// TIA Portal project "PHASE2_Final_Team2 Final W HMI" (V16)

(* hardware
DEVICE "S71500/ET200MP station_1"  S7-1500 station
   slot 0: "Rail_0"  Rack  6ES7 590-1***0-0AA0
   slot 1: "PLC_1"  CPU 1513-1 PN  6ES7 513-1AL02-0AB0  V2.8
      slot 3: "CPU display_1"  6ES7591-1AA00-0AA0
      slot 32768: "PROFINET interface_1"  X1
         slot 32769: "Port_1"  X1 P1
         slot 32770: "Port_2"  X1 P2
      slot 34817: "Virtual CP interface port_1"  Virtual CP interface port  Virtual CP interface port
   slot 2: "DI 16x24VDC BA_1"  DI 16x24VDC BA  6ES7 521-1BH10-0AA0  V1.1
   slot 3: "DQ 16x24VDC/0.5A BA_1"  DQ 16x24VDC/0.5A BA  6ES7 522-1BH10-0AA0  V1.1
DEVICE "HMI_1"  TP700 Comfort
   slot 0: "HMI_1"  TP700 Comfort  6AV2 124-0GC01-0AX0  16.0.0.0
   slot 1: "HMI_RT_1"  TP700 Comfort  6AV2 124-0GC01-0AX0  16.0.0.0
   slot 5: "HMI_1.IE_CP_1"  PROFINET Interface  16.0.0.0
      slot 1: "PROFINET Interface_1"  PROFINET Interface
         slot 1: "Port_1"  Port
         slot 2: "Port_2"  Port
   slot 7: "HMI_1.MPI/DP_CP_1"  MPI/DP Interface  16.0.0.0
*)

// ===== PLC "PLC_1"  CPU 1513-1 PN =====

VAR_GLOBAL   // PLC tag table "Default tag table"
   "start whole system" AT %I3.1 : Bool;
   "stop whole system" AT %I3.2 : Bool;
   "Lid Exit Stop" AT %M251.0 : Bool;
   "LID exit Stop Sensor" AT %I7.2 : Bool;
   "Base Exit Stop Sensor" AT %I7.1 : Bool;
   "Base Exit Stop" AT %M250.0 : Bool;
END_VAR

VAR_GLOBAL   // PLC tag table "pick&place"
   "Item_at_entry" AT %I0.0 : Bool;
   "Item at Exit" AT %I0.1 : Bool;
   "Moving X" AT %M171.0 : Bool;
   "Moving Z" AT %M170.0 : Bool;
   "Item Detected" AT %I0.2 : Bool;
   "Start Button" AT %I0.3 : Bool;
   "Reset" AT %I0.4 : Bool;
   "Stop" AT %I0.5 : Bool;
   "Emergency stop" AT %I0.6 : Bool;
   "Entry_conveyor" AT %Q5.0 : Bool;
   "Exit conveyor" AT %Q5.1 : Bool;
   "Move X" AT %Q5.2 : Bool;
   "Move Z" AT %Q12.3 : Bool;
   "Grab" AT %Q0.4 : Bool;
   "Start light 1" AT %Q4.5 : Bool;
   "Reset light 1" AT %Q5.6 : Bool;
   "Stop light 1" AT %Q0.7 : Bool;
   "s1" AT %M92.0 : Bool;
   "s2" AT %M93.0 : Bool;
   "s3" AT %M94.0 : Bool;
   "s4" AT %M95.0 : Bool;
   "s5" AT %M96.0 : Bool;
   "s6" AT %M97.0 : Bool;
   "s7" AT %M98.0 : Bool;
   "s8" AT %M99.0 : Bool;
   "Entry Conveyor 1" AT %QD30 : Real;
   "Exit_Conveyor 1" AT %QD34 : Real;
   "Move_X 1" AT %QD38 : Real;
   "Move_Z 1" AT %QD42 : Real;
   "Moving_X 1" AT %ID30 : Real;
   "Moving_Z 1" AT %ID34 : Real;
   "Item_at_entry(1)" AT %I0.7 : Bool;
   "Item at Exit(1)" AT %I1.0 : Bool;
   "Moving X(1)" AT %M172.0 : Bool;
   "Moving Z(1)" AT %M173.0 : Bool;
   "Item Detected(1)" AT %I1.1 : Bool;
   "Start Button(1)" AT %I1.2 : Bool;
   "Reset(1)" AT %I1.3 : Bool;
   "Stop(1)" AT %I1.4 : Bool;
   "Emergency stop(1)" AT %I1.5 : Bool;
   "Entry_conveyor(1)" AT %M120.0 : Bool;
   "Exit conveyor(1)" AT %Q7.1 : Bool;
   "Move X(1)" AT %Q7.2 : Bool;
   "Move Z(1)" AT %Q7.3 : Bool;
   "Grab(1)" AT %Q0.5 : Bool;
   "Start light 1(1)" AT %Q3.5 : Bool;
   "Reset light 1(1)" AT %Q3.6 : Bool;
   "Stop light 1(1)" AT %Q3.7 : Bool;
   "Counter 1(1)" AT %QD60 : DInt;
   "s1(1)" AT %M14.0 : Bool;
   "s2(1)" AT %M101.0 : Bool;
   "s3(1)" AT %M102.0 : Bool;
   "s4(1)" AT %M103.0 : Bool;
   "s5(1)" AT %M104.0 : Bool;
   "s6(1)" AT %M105.0 : Bool;
   "s7(1)" AT %M106.0 : Bool;
   "s8(1)" AT %M107.0 : Bool;
   "Entry Conveyor 1(1)" AT %QD46 : Real;
   "Exit_Conveyor 1(1)" AT %QD50 : Real;
   "Move_X 1(1)" AT %QD54 : Real;
   "Move_Z 1(1)" AT %QD58 : Real;
   "Moving_X 1(1)" AT %ID38 : Real;
   "Moving_Z 1(1)" AT %ID42 : Real;
   "Emitter 1" AT %Q2.2 : Bool;
   "Emitter 0" AT %Q2.3 : Bool;
END_VAR

VAR_GLOBAL   // PLC tag table "machine_center"
   "Start_System" AT %I2.6 : Bool;
   "Stop_System" AT %I2.7 : Bool;
   "Lids_Raw_conveyor" AT %M72.0 : Bool;
   "Bases_raw_conveyor" AT %M73.0 : Bool;
   "S1(2)" AT %M100.0 : Bool;
   "S2(2)" AT %M108.0 : Bool;
   "S3(2)" AT %M109.0 : Bool;
   "S4(2)" AT %M110.0 : Bool;
   "S5(2)" AT %M111.0 : Bool;
   "S6(2)" AT %M112.0 : Bool;
   "S7(2)" AT %M113.0 : Bool;
   "S8(2)" AT %M8.0 : Bool;
   "S9" AT %M9.0 : Bool;
   "S10" AT %M10.0 : Bool;
   "Emergency Stop System" AT %I3.0 : Bool;
   "Start_Light" AT %Q1.1 : Bool;
   "Stop_lights" AT %Q1.2 : Bool;
   "Lids_at_entry" AT %I1.6 : Bool;
   "Bases At entry" AT %I2.2 : Bool;
   "Lids_center_busy" AT %I1.7 : Bool;
   "Lids_at_exit" AT %I2.1 : Bool;
   "Lids_center_error" AT %I2.0 : Bool;
   "Bases_at_exit" AT %I2.5 : Bool;
   "bases_center_busy" AT %I2.3 : Bool;
   "Base_center_error" AT %I2.4 : Bool;
   "S11" AT %M11.0 : Bool;
   "S12" AT %M12.0 : Bool;
   "Exit_Conveyor" AT %Q11.6 : Bool;
   "Produce_Lids" AT %Q0.0 : Bool;
   "Lids_Center_Start" AT %Q0.1 : Bool;
   "Bases_center_start" AT %Q0.6 : Bool;
   "Reset_Lids" AT %Q0.2 : Bool;
   "Stop_Lids" AT %Q0.3 : Bool;
   "Reset_Base" AT %Q10.6 : Bool;
   "Stop_Bases" AT %Q10.7 : Bool;
   "Lids_Exit_convyor1" AT %M70.0 : Bool;
   "LIDS Sorting Conveyor1" AT %M71.0 : Bool;
   "Bases_Exit_conveyor1" AT %M206.0 : Bool;
   "Bases Sorting Conveyor" AT %M205.0 : Bool;
   "Lids_Count" AT %QW10 : Int;
   "Bases_Count" AT %QW20 : Int;
   "Tag_1" AT %M13.0 : Bool;
   "S13" AT %M64.0 : Bool;
   "S14" AT %M65.0 : Bool;
   "Tag_2" AT %M66.0 : Bool;
   "Tag_3" AT %M67.0 : Bool;
   "Lids_Arrived" AT %I11.5 : Bool;
   "Bases Arrived" AT %I11.4 : Bool;
   "LIDS_RAW_CONVEYOR_aNALOG" AT %QD62 : Real;
   "Lid_exit_conveyor1_analog" AT %QD66 : Real;
   "Base_raw_conveyor_analog" AT %QD70 : Real;
   "Base_exit_conveyor1_analog" AT %QD74 : Real;
END_VAR

VAR_GLOBAL   // PLC tag table "Sorting"
   "Bases Sorter turn" AT %Q1.5 : Bool;
   "bases Sorter  Belt" AT %Q1.6 : Bool;
   "LID sorter Turn" AT %Q1.3 : Bool;
   "LID sorter Belt" AT %Q1.4 : Bool;
   "Base Sorting Sensor" AT %ID50 : DWord;
   "Base_Exit_conveyor_blue" AT %M84.0 : Bool;
   "Vision sensor in range" AT %Q46.4 : Bool;
   "Stop Entry conveyor" AT %Q46.5 : Bool;
   "Blue lid" AT %M200.0 : Bool;
   "Green lid" AT %M201.0 : Bool;
   "Tag_1(1)" AT %M50.0 : Bool;
   "Tag_2(1)" AT %M51.0 : Bool;
   "S1(3)" AT %M52.0 : Bool;
   "S2(3)" AT %M53.0 : Bool;
   "S3(3)" AT %M54.0 : Bool;
   "S4(3)" AT %M55.0 : Bool;
   "S5(3)" AT %M56.0 : Bool;
   "S6(3)" AT %M57.0 : Bool;
   "S1(4)" AT %M58.0 : Bool;
   "S2(4)" AT %M59.0 : Bool;
   "S3(4)" AT %M60.0 : Bool;
   "S5(4)" AT %M61.0 : Bool;
   "S4(4)" AT %M62.0 : Bool;
   "S6(4)" AT %M63.0 : Bool;
   "Base Start Sorting" AT %I4.0 : Bool;
   "Base Exit Conveyor Green" AT %M85.0 : Bool;
   "Bases Blue Sorted Conv" AT %QD106 : Real;
   "Bases Green Sorted Conv" AT %QD102 : Real;
   "LID Start Sorting" AT %I3.7 : Bool;
   "LID sorting Sensor" AT %ID46 : DWord;
   "LIDs_Blue_Sorted_conv" AT %M86.0 : Bool;
   "LIDs green sorted conv" AT %M87.0 : Bool;
   "LID blue sorted conv ana" AT %QD98 : Real;
   "LID green Sorted Conv ANalog" AT %QD94 : Real;
   "Emergency Stop Base" AT %I4.1 : Bool;
   "Emergency Stop LID" AT %I4.2 : Bool;
   "Blue Base" AT %M90.0 : Bool;
   "Green Base" AT %M91.0 : Bool;
   "LID Green Sorted" AT %I3.4 : Bool;
   "LID Blue Sorted" AT %I3.3 : Bool;
   "LIDS sorting Conveyor 2" AT %M82.0 : Bool;
   "Base Blue Sorted" AT %I3.5 : Bool;
   "Base Green Sorted" AT %I3.6 : Bool;
   "Curved Bases Sorting Conveyor" AT %M83.0 : Bool;
   "LID sorting conveyor 1" AT %QD78 : Real;
   "LID Sorting Conveyor 2" AT %QD82 : Real;
   "Base Sorting Conveyor" AT %QD86 : Real;
   "Curved Base Sorting Conveyor" AT %QD90 : Real;
   "LID green Sorted Conv ANalog(1)" AT %QD110 : Real;
   "LID green Sorted Conv ANalog(2)" AT %QD114 : Real;
   "LID green Sorted Conv ANalog(3)" AT %QD118 : Real;
   "LID blue sorted conv ana(1)" AT %QD122 : Real;
   "LID blue sorted conv ana(2)" AT %QD126 : Real;
   "Bases Blue Sorted Conv(1)" AT %QD130 : Real;
   "Bases Blue Sorted Conv(2)" AT %QD134 : Real;
   "Bases Green Sorted Conv(1)" AT %QD138 : Real;
   "Bases Green Sorted Conv(2)" AT %QD142 : Real;
   "Bases Green Sorted Conv(3)" AT %QD146 : Real;
   "Bases Green Sorted Conv(4)" AT %QD150 : Real;
   "Bases Green Sorted Conv(5)" AT %QD154 : Real;
   "Bases Green Sorted Conv(6)" AT %QD158 : Real;
END_VAR

VAR_GLOBAL   // PLC tag table "BlueAssembler"
   "S1(7) Blue Assembler" AT %M121.0 : Bool;
   "S2(7) Blue Assembler" AT %M122.0 : Bool;
   "S3(7) Blue Assembler" AT %M123.0 : Bool;
   "S4(7) Blue Assembler" AT %M124.0 : Bool;
   "S5(7) Blue Assembler" AT %M125.0 : Bool;
   "S6(7) Blue Assembler" AT %M126.0 : Bool;
   "S7(5) Blue Assembler" AT %M127.0 : Bool;
   "S8(5) Blue Assembler" AT %M128.0 : Bool;
   "S9(1) Blue Assembler" AT %M129.0 : Bool;
   "Emergency Stop Blue Assembler" AT %I5.3 : Bool;
   "Lid at place Blue Assembler" AT %I4.6 : Bool;
   "base at place Blue Assembler" AT %I5.0 : Bool;
   "Lid_clamped Blue Assembler" AT %I4.7 : Bool;
   "Item Detected Blue Assembler" AT %I4.5 : Bool;
   "Moving_z Blue Assembler" AT %I4.4 : Bool;
   "Tag_1(2) Blue Assembler" AT %M139.0 : Bool;
   "Base Clamped Blue Assembler" AT %I5.1 : Bool;
   "Tag_2(2) Blue Assembler" AT %M140.0 : Bool;
   "Moving_X Blue Assembler" AT %I4.3 : Bool;
   "Tag_3(1) Blue Assembler" AT %M141.0 : Bool;
   "Tag_4 Blue Assembler" AT %M142.0 : Bool;
   "Part_leaving Blue Assembler" AT %I5.2 : Bool;
   "S10(1) Blue Assembler" AT %M143.0 : Bool;
   "Tag_5 Blue Assembler" AT %M144.0 : Bool;
   "Lid _ Conveyor Blue Assembler" AT %M151.0 : Bool;
   "Bases Conveyor Blue Assembler" AT %M152.0 : Bool;
   "Clamp-base Blue Assembler" AT %Q2.5 : Bool;
   "Clamp_lid Blue Assembler" AT %Q2.6 : Bool;
   "grab Blue Assembler" AT %Q2.4 : Bool;
   "Pos_raise_bases Blue Assembler" AT %Q2.7 : Bool;
   "Tag_6Blue Assembler" AT %M147.0 : Bool;
   "S11(1) Blue Assembler" AT %M150.0 : Bool;
   "Tag_7Blue Assembler" AT %M145.0 : Bool;
   "Tag_8Blue Assembler" AT %M146.0 : Bool;
   "Lid_Conveyor_Analog Blue Assembler" AT %QD162 : Real;
   "Base_Conveyor_analog Blue Assembler" AT %QD166 : Real;
   "move_xBlue Assembler" AT %M148.0 : Bool;
   "Move_X_analog Blue Assembler" AT %QD170 : Real;
   "move_z Blue Assembler" AT %M149.0 : Bool;
   "Move_Z_analog Blue Assembler" AT %QD174 : Real;
   "Start base BlueAssembly(1)" AT %I5.4 : Bool;
   "Start LID Blue Assembly(1)" AT %I5.5 : Bool;
END_VAR

VAR_GLOBAL   // PLC tag table "GreenAssembler"
   "S1(8) Green" AT %M130.0 : Bool;
   "S2(8) Green" AT %M131.0 : Bool;
   "S3(8) Green" AT %M132.0 : Bool;
   "S4(8) Green" AT %M133.0 : Bool;
   "S5(8) Green" AT %M134.0 : Bool;
   "S6(8) Green" AT %M135.0 : Bool;
   "S7(6) Green" AT %M136.0 : Bool;
   "S8(6) Green" AT %M137.0 : Bool;
   "S9(2) Green" AT %M138.0 : Bool;
   "Emergency Stop Green assembler" AT %I6.6 : Bool;
   "Lid at place(1) Green" AT %I6.1 : Bool;
   "base at place(1) Green" AT %I6.3 : Bool;
   "Lid_clamped(1) Green" AT %I6.2 : Bool;
   "Item Detected(3) Green" AT %I6.0 : Bool;
   "Moving_z(1) Green" AT %I5.7 : Bool;
   "Tag_1(3) Green" AT %M153.0 : Bool;
   "Base Clamped(1) Green" AT %I6.4 : Bool;
   "Tag_2(3) Green" AT %M154.0 : Bool;
   "Moving_X Green" AT %I5.6 : Bool;
   "Tag_3(2) Green" AT %M155.0 : Bool;
   "Tag_4(1) Green" AT %M156.0 : Bool;
   "Part_leaving(1) Green" AT %I6.5 : Bool;
   "S10(2) Green" AT %M157.0 : Bool;
   "Tag_5(1) Green" AT %M158.0 : Bool;
   "Lid _ Conveyor(1) Green" AT %M165.0 : Bool;
   "Bases Conveyor(1) Green" AT %M166.0 : Bool;
   "Clamp-base(1) Green" AT %Q3.1 : Bool;
   "Clamp_lid(1) Green" AT %Q3.2 : Bool;
   "grab(4) Green" AT %Q3.0 : Bool;
   "Pos_raise_bases(1) Green" AT %Q3.3 : Bool;
   "Tag_6(1) Green" AT %M161.0 : Bool;
   "S11(2) Green" AT %M164.0 : Bool;
   "Tag_7(1) Green" AT %M159.0 : Bool;
   "Tag_8(1) Green" AT %M160.0 : Bool;
   "Lid_Conveyor_Analog(1) Green" AT %QD178 : Real;
   "Base_Conveyor_analog(1) Green" AT %QD182 : Real;
   "move_x(1) Green" AT %M162.0 : Bool;
   "Move_X_analog(1) Green" AT %QD186 : Real;
   "move_z(1) Green" AT %M163.0 : Bool;
   "Move_Z_analog(1) Green" AT %QD190 : Real;
   "Start base Green Assembly" AT %I6.7 : Bool;
   "Start LID Green Assembly" AT %I7.0 : Bool;
END_VAR

DATA_BLOCK "machine_center_DB"   // DB1
{ S7_Optimized_Access := 'TRUE' }
VERSION : 0.1
// stored: InstanceOfName machine_center
"machine_center"
BEGIN
END_DATA_BLOCK

DATA_BLOCK "Sorting2_DB"   // DB2
{ S7_Optimized_Access := 'TRUE' }
VERSION : 0.1
// stored: InstanceOfName Sorting2
"Sorting2"
BEGIN
END_DATA_BLOCK

DATA_BLOCK "Pick&Place1_DB"   // DB3
{ S7_Optimized_Access := 'TRUE' }
VERSION : 0.1
// stored: InstanceOfName Pick&Place1
"Pick&Place1"
BEGIN
END_DATA_BLOCK

DATA_BLOCK "Pick&Place2_DB"   // DB4
{ S7_Optimized_Access := 'TRUE' }
VERSION : 0.1
// stored: InstanceOfName Pick&Place2
"Pick&Place2"
BEGIN
END_DATA_BLOCK

DATA_BLOCK "Sorting1_DB"   // DB5
{ S7_Optimized_Access := 'TRUE' }
VERSION : 0.1
// stored: InstanceOfName Sorting1
"Sorting1"
BEGIN
END_DATA_BLOCK

DATA_BLOCK "Assembler Blue_DB"   // DB6
{ S7_Optimized_Access := 'TRUE' }
VERSION : 0.1
// stored: InstanceOfName Assembler Blue
"Assembler Blue"
BEGIN
END_DATA_BLOCK

DATA_BLOCK "Assembler Green_DB"   // DB7
{ S7_Optimized_Access := 'TRUE' }
VERSION : 0.1
// stored: InstanceOfName Assembler Green
"Assembler Green"
BEGIN
END_DATA_BLOCK

DATA_BLOCK "HMI_Area_Pointer"   // DB8
{ S7_Optimized_Access := 'TRUE' }
VERSION : 0.1
   VAR
      "Job MailBox" : Array[0..3] of Word;
      NumScreen : Int;
      "Start Whole System PB" : Bool;
      "Stop Whole System PB" : Bool;
      HMI_Box_Pick_and_place1 : DWord := 0;
      HMI_Box_Pick_and_place2 : DWord := 0;
      "HMI blue part sorted move HMI" : DWord := 0;
      "HMI Green part sorted move HMI" : DWord := 0;
   END_VAR
BEGIN
   "Job MailBox"[0] := 51;
   "Job MailBox"[2] := 0;
   "Job MailBox"[3] := 0;
END_DATA_BLOCK

// folder: System blocks/Program resources

DATA_BLOCK "IEC_Timer_0_DB"   // DB9
{ S7_Optimized_Access := 'TRUE' }
AUTHOR : Simatic
FAMILY : IEC
NAME : IEC_TMR
VERSION : 1.0
// stored: InstanceOfName IEC_TIMER
"IEC_TIMER"
BEGIN
END_DATA_BLOCK

DATA_BLOCK "IEC_Timer_0_DB_1"   // DB10
{ S7_Optimized_Access := 'TRUE' }
AUTHOR : Simatic
FAMILY : IEC
NAME : IEC_TMR
VERSION : 1.0
// stored: InstanceOfName IEC_TIMER
"IEC_TIMER"
BEGIN
END_DATA_BLOCK

DATA_BLOCK "IEC_Timer_0_DB_2"   // DB11
{ S7_Optimized_Access := 'TRUE' }
AUTHOR : Simatic
FAMILY : IEC
NAME : IEC_TMR
VERSION : 1.0
// stored: InstanceOfName IEC_TIMER
"IEC_TIMER"
BEGIN
END_DATA_BLOCK

DATA_BLOCK "IEC_Timer_0_DB_3"   // DB12
{ S7_Optimized_Access := 'TRUE' }
AUTHOR : Simatic
FAMILY : IEC
NAME : IEC_TMR
VERSION : 1.0
// stored: InstanceOfName IEC_TIMER
"IEC_TIMER"
BEGIN
END_DATA_BLOCK

// folder: (top level)

FUNCTION_BLOCK "Pick&Place1"   // FB1, LAD
{ S7_Optimized_Access := 'TRUE' }
VERSION : 0.1
BEGIN

REGION Network 1
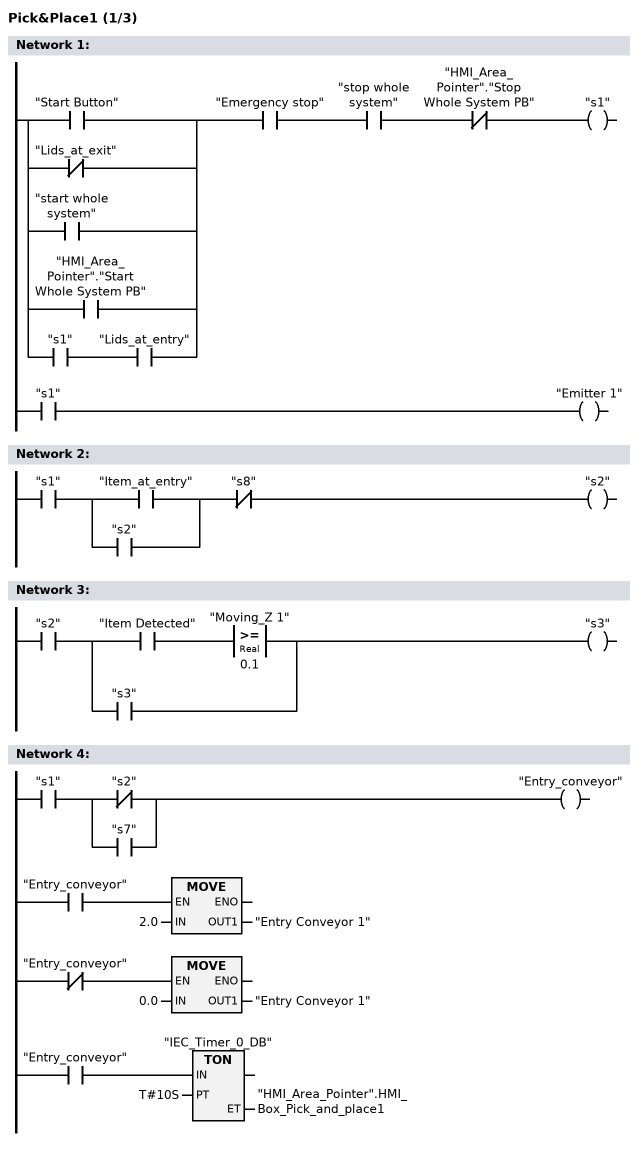
   RUNG wire#powerrail
      Contact( "Start Button" )
      wire#w1
      Contact( "Emergency stop" )
      Contact( "stop whole system" )
      I_Contact( "HMI_Area_Pointer"."Stop Whole System PB" )
      Coil( "s1" )
   END_RUNG
   RUNG wire#powerrail
      I_Contact( "Lids_at_exit" )
   END_RUNG wire#w1
   RUNG wire#powerrail
      Contact( "start whole system" )
   END_RUNG wire#w1
   RUNG wire#powerrail
      Contact( "HMI_Area_Pointer"."Start Whole System PB" )
   END_RUNG wire#w1
   RUNG wire#powerrail
      Contact( "s1" )
      Contact( "Lids_at_entry" )
   END_RUNG wire#w1
   RUNG wire#powerrail
      Contact( "s1" )
      Coil( "Emitter 1" )
   END_RUNG
   // the same network as SCL:
   "s1" := ("Start Button" OR NOT "Lids_at_exit" OR "start whole system" OR "HMI_Area_Pointer"."Start Whole System PB" OR ("s1" AND "Lids_at_entry")) AND "Emergency stop" AND "stop whole system" AND NOT "HMI_Area_Pointer"."Stop Whole System PB";
   "Emitter 1" := "s1";
END_REGION

REGION Network 2
   RUNG wire#powerrail
      Contact( "s1" )
      wire#w1
      Contact( "Item_at_entry" )
      wire#w2
      I_Contact( "s8" )
      Coil( "s2" )
   END_RUNG
   RUNG wire#w1
      Contact( "s2" )
   END_RUNG wire#w2
   // the same network as SCL:
   "s2" := "s1" AND ("Item_at_entry" OR "s2") AND NOT "s8";
END_REGION

REGION Network 3
   RUNG wire#powerrail
      Contact( "s2" )
      wire#w1
      Contact( "Item Detected" )
      { S7_Templates := "SrcType := Real" } GE_Contact(in1 := "Moving_Z 1", in2 := 0.1)
      wire#w2
      Coil( "s3" )
   END_RUNG
   RUNG wire#w1
      Contact( "s3" )
   END_RUNG wire#w2
   // the same network as SCL:
   "s3" := "s2" AND (("Item Detected" AND ("Moving_Z 1" >= 0.1)) OR "s3");
END_REGION

REGION Network 4
   "Entry_conveyor" := "s1" AND (NOT "s2" OR "s7");
   IF "Entry_conveyor" THEN "Entry Conveyor 1" := 2.0; END_IF;
   IF NOT "Entry_conveyor" THEN "Entry Conveyor 1" := 0.0; END_IF;
   "IEC_Timer_0_DB".TON(IN := "Entry_conveyor", PT := T#10S, ET => "HMI_Area_Pointer".HMI_Box_Pick_and_place1);
END_REGION

REGION Network 5
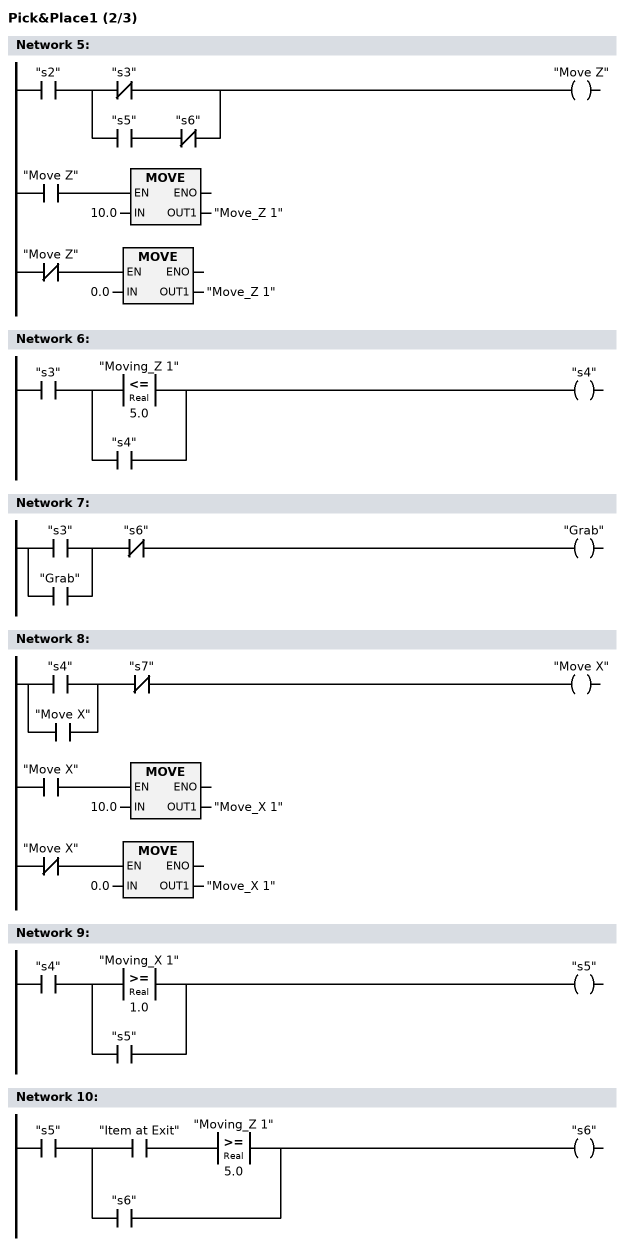
   RUNG wire#powerrail
      Contact( "s2" )
      wire#w1
      I_Contact( "s3" )
      wire#w2
      Coil( "Move Z" )
   END_RUNG
   RUNG wire#w1
      Contact( "s5" )
      I_Contact( "s6" )
   END_RUNG wire#w2
   RUNG wire#powerrail
      Contact( "Move Z" )
      Move(in := 10.0, out1 => "Move_Z 1")
   END_RUNG
   RUNG wire#powerrail
      I_Contact( "Move Z" )
      Move(in := 0.0, out1 => "Move_Z 1")
   END_RUNG
   // the same network as SCL:
   "Move Z" := "s2" AND (NOT "s3" OR ("s5" AND NOT "s6"));
   IF "Move Z" THEN "Move_Z 1" := 10.0; END_IF;
   IF NOT "Move Z" THEN "Move_Z 1" := 0.0; END_IF;
END_REGION

REGION Network 6
   RUNG wire#powerrail
      Contact( "s3" )
      wire#w1
      { S7_Templates := "SrcType := Real" } LE_Contact(in1 := "Moving_Z 1", in2 := 5.0)
      wire#w2
      Coil( "s4" )
   END_RUNG
   RUNG wire#w1
      Contact( "s4" )
   END_RUNG wire#w2
   // the same network as SCL:
   "s4" := "s3" AND (("Moving_Z 1" <= 5.0) OR "s4");
END_REGION

REGION Network 7
   RUNG wire#powerrail
      Contact( "s3" )
      wire#w1
      I_Contact( "s6" )
      Coil( "Grab" )
   END_RUNG
   RUNG wire#powerrail
      Contact( "Grab" )
   END_RUNG wire#w1
   // the same network as SCL:
   "Grab" := ("s3" OR "Grab") AND NOT "s6";
END_REGION

REGION Network 8
   RUNG wire#powerrail
      Contact( "s4" )
      wire#w1
      I_Contact( "s7" )
      Coil( "Move X" )
   END_RUNG
   RUNG wire#powerrail
      Contact( "Move X" )
   END_RUNG wire#w1
   RUNG wire#powerrail
      Contact( "Move X" )
      Move(in := 10.0, out1 => "Move_X 1")
   END_RUNG
   RUNG wire#powerrail
      I_Contact( "Move X" )
      Move(in := 0.0, out1 => "Move_X 1")
   END_RUNG
   // the same network as SCL:
   "Move X" := ("s4" OR "Move X") AND NOT "s7";
   IF "Move X" THEN "Move_X 1" := 10.0; END_IF;
   IF NOT "Move X" THEN "Move_X 1" := 0.0; END_IF;
END_REGION

REGION Network 9
   RUNG wire#powerrail
      Contact( "s4" )
      wire#w1
      { S7_Templates := "SrcType := Real" } GE_Contact(in1 := "Moving_X 1", in2 := 1.0)
      wire#w2
      Coil( "s5" )
   END_RUNG
   RUNG wire#w1
      Contact( "s5" )
   END_RUNG wire#w2
   // the same network as SCL:
   "s5" := "s4" AND (("Moving_X 1" >= 1.0) OR "s5");
END_REGION

REGION Network 10
   RUNG wire#powerrail
      Contact( "s5" )
      wire#w1
      Contact( "Item at Exit" )
      { S7_Templates := "SrcType := Real" } GE_Contact(in1 := "Moving_Z 1", in2 := 5.0)
      wire#w2
      Coil( "s6" )
   END_RUNG
   RUNG wire#w1
      Contact( "s6" )
   END_RUNG wire#w2
   // the same network as SCL:
   "s6" := "s5" AND (("Item at Exit" AND ("Moving_Z 1" >= 5.0)) OR "s6");
END_REGION

REGION Network 11
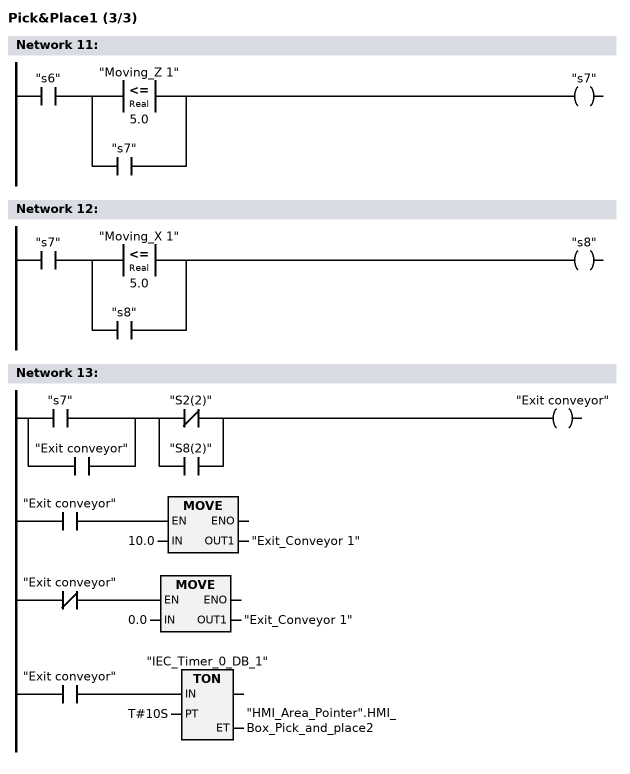
   RUNG wire#powerrail
      Contact( "s6" )
      wire#w1
      { S7_Templates := "SrcType := Real" } LE_Contact(in1 := "Moving_Z 1", in2 := 5.0)
      wire#w2
      Coil( "s7" )
   END_RUNG
   RUNG wire#w1
      Contact( "s7" )
   END_RUNG wire#w2
   // the same network as SCL:
   "s7" := "s6" AND (("Moving_Z 1" <= 5.0) OR "s7");
END_REGION

REGION Network 12
   RUNG wire#powerrail
      Contact( "s7" )
      wire#w1
      { S7_Templates := "SrcType := Real" } LE_Contact(in1 := "Moving_X 1", in2 := 5.0)
      wire#w2
      Coil( "s8" )
   END_RUNG
   RUNG wire#w1
      Contact( "s8" )
   END_RUNG wire#w2
   // the same network as SCL:
   "s8" := "s7" AND (("Moving_X 1" <= 5.0) OR "s8");
END_REGION

REGION Network 13
   "Exit conveyor" := ("s7" OR "Exit conveyor") AND (NOT "S2(2)" OR "S8(2)");
   IF "Exit conveyor" THEN "Exit_Conveyor 1" := 10.0; END_IF;
   IF NOT "Exit conveyor" THEN "Exit_Conveyor 1" := 0.0; END_IF;
   "IEC_Timer_0_DB_1".TON(IN := "Exit conveyor", PT := T#10S, ET => "HMI_Area_Pointer".HMI_Box_Pick_and_place2);
END_REGION
END_FUNCTION_BLOCK

FUNCTION_BLOCK "Pick&Place2"   // FB2, LAD
{ S7_Optimized_Access := 'TRUE' }
VERSION : 0.1
BEGIN

REGION Network 1
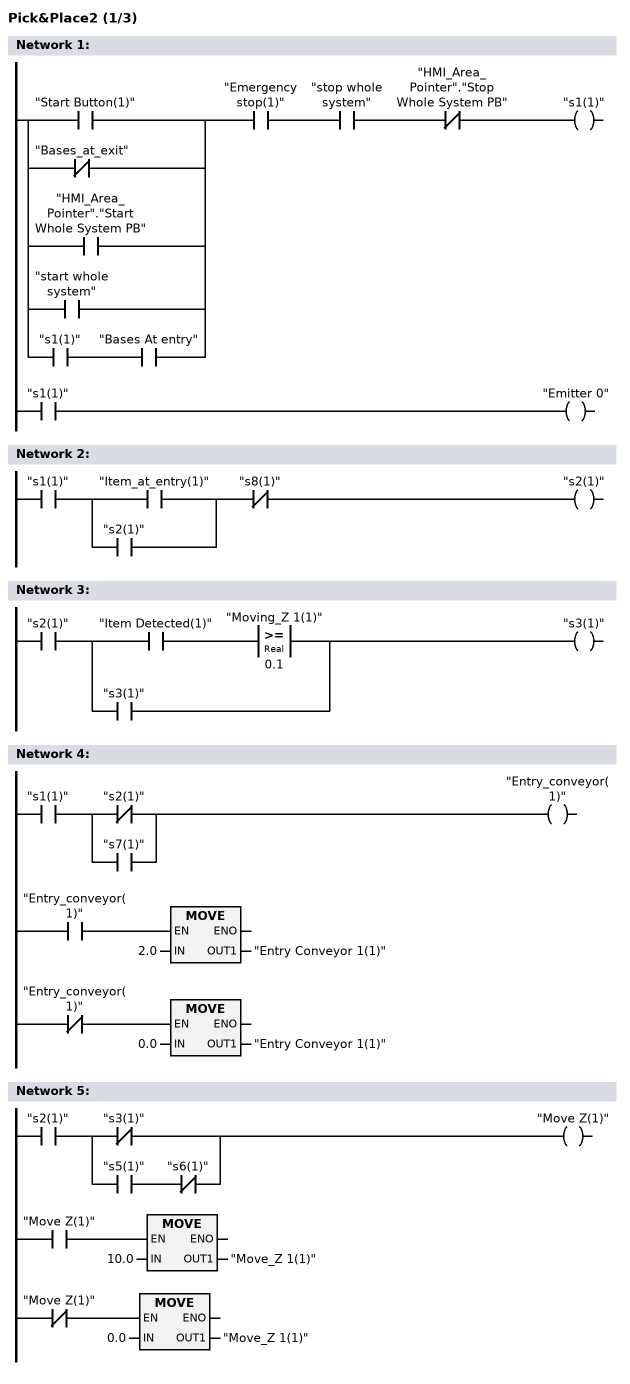
   RUNG wire#powerrail
      Contact( "Start Button(1)" )
      wire#w1
      Contact( "Emergency stop(1)" )
      Contact( "stop whole system" )
      I_Contact( "HMI_Area_Pointer"."Stop Whole System PB" )
      Coil( "s1(1)" )
   END_RUNG
   RUNG wire#powerrail
      I_Contact( "Bases_at_exit" )
   END_RUNG wire#w1
   RUNG wire#powerrail
      Contact( "HMI_Area_Pointer"."Start Whole System PB" )
   END_RUNG wire#w1
   RUNG wire#powerrail
      Contact( "start whole system" )
   END_RUNG wire#w1
   RUNG wire#powerrail
      Contact( "s1(1)" )
      Contact( "Bases At entry" )
   END_RUNG wire#w1
   RUNG wire#powerrail
      Contact( "s1(1)" )
      Coil( "Emitter 0" )
   END_RUNG
   // the same network as SCL:
   "s1(1)" := ("Start Button(1)" OR NOT "Bases_at_exit" OR "HMI_Area_Pointer"."Start Whole System PB" OR "start whole system" OR ("s1(1)" AND "Bases At entry")) AND "Emergency stop(1)" AND "stop whole system" AND NOT "HMI_Area_Pointer"."Stop Whole System PB";
   "Emitter 0" := "s1(1)";
END_REGION

REGION Network 2
   RUNG wire#powerrail
      Contact( "s1(1)" )
      wire#w1
      Contact( "Item_at_entry(1)" )
      wire#w2
      I_Contact( "s8(1)" )
      Coil( "s2(1)" )
   END_RUNG
   RUNG wire#w1
      Contact( "s2(1)" )
   END_RUNG wire#w2
   // the same network as SCL:
   "s2(1)" := "s1(1)" AND ("Item_at_entry(1)" OR "s2(1)") AND NOT "s8(1)";
END_REGION

REGION Network 3
   RUNG wire#powerrail
      Contact( "s2(1)" )
      wire#w1
      Contact( "Item Detected(1)" )
      { S7_Templates := "SrcType := Real" } GE_Contact(in1 := "Moving_Z 1(1)", in2 := 0.1)
      wire#w2
      Coil( "s3(1)" )
   END_RUNG
   RUNG wire#w1
      Contact( "s3(1)" )
   END_RUNG wire#w2
   // the same network as SCL:
   "s3(1)" := "s2(1)" AND (("Item Detected(1)" AND ("Moving_Z 1(1)" >= 0.1)) OR "s3(1)");
END_REGION

REGION Network 4
   RUNG wire#powerrail
      Contact( "s1(1)" )
      wire#w1
      I_Contact( "s2(1)" )
      wire#w2
      Coil( "Entry_conveyor(1)" )
   END_RUNG
   RUNG wire#w1
      Contact( "s7(1)" )
   END_RUNG wire#w2
   RUNG wire#powerrail
      Contact( "Entry_conveyor(1)" )
      Move(in := 2.0, out1 => "Entry Conveyor 1(1)")
   END_RUNG
   RUNG wire#powerrail
      I_Contact( "Entry_conveyor(1)" )
      Move(in := 0.0, out1 => "Entry Conveyor 1(1)")
   END_RUNG
   // the same network as SCL:
   "Entry_conveyor(1)" := "s1(1)" AND (NOT "s2(1)" OR "s7(1)");
   IF "Entry_conveyor(1)" THEN "Entry Conveyor 1(1)" := 2.0; END_IF;
   IF NOT "Entry_conveyor(1)" THEN "Entry Conveyor 1(1)" := 0.0; END_IF;
END_REGION

REGION Network 5
   RUNG wire#powerrail
      Contact( "s2(1)" )
      wire#w1
      I_Contact( "s3(1)" )
      wire#w2
      Coil( "Move Z(1)" )
   END_RUNG
   RUNG wire#w1
      Contact( "s5(1)" )
      I_Contact( "s6(1)" )
   END_RUNG wire#w2
   RUNG wire#powerrail
      Contact( "Move Z(1)" )
      Move(in := 10.0, out1 => "Move_Z 1(1)")
   END_RUNG
   RUNG wire#powerrail
      I_Contact( "Move Z(1)" )
      Move(in := 0.0, out1 => "Move_Z 1(1)")
   END_RUNG
   // the same network as SCL:
   "Move Z(1)" := "s2(1)" AND (NOT "s3(1)" OR ("s5(1)" AND NOT "s6(1)"));
   IF "Move Z(1)" THEN "Move_Z 1(1)" := 10.0; END_IF;
   IF NOT "Move Z(1)" THEN "Move_Z 1(1)" := 0.0; END_IF;
END_REGION

REGION Network 6
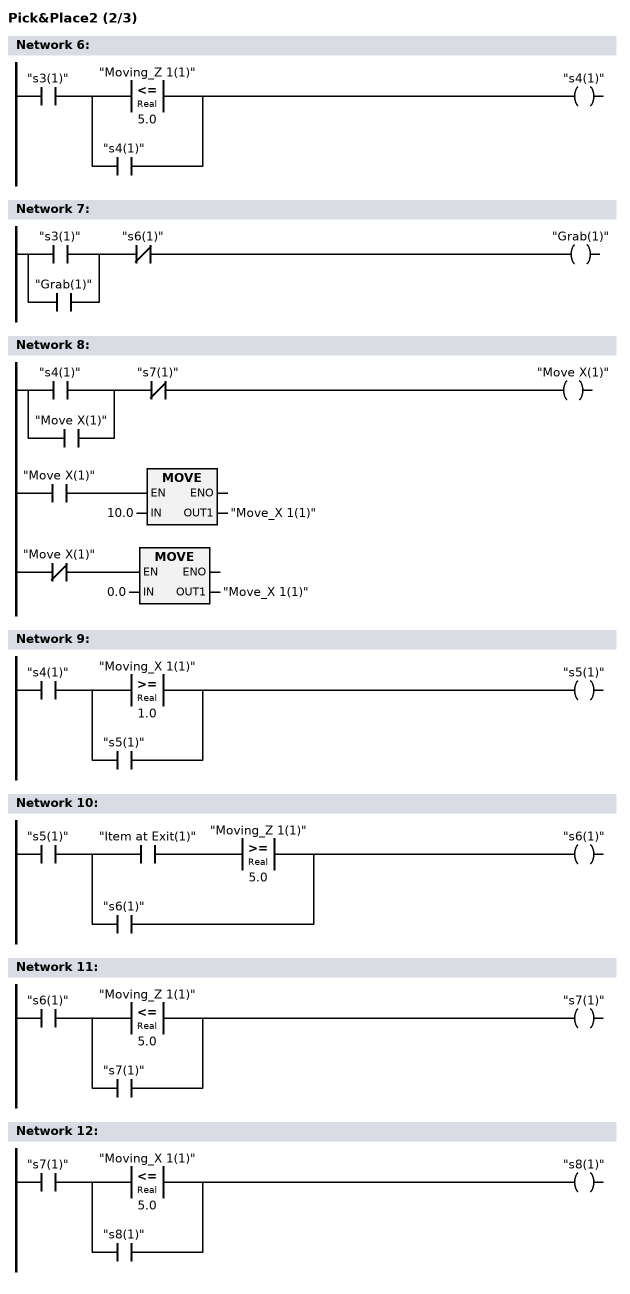
   RUNG wire#powerrail
      Contact( "s3(1)" )
      wire#w1
      { S7_Templates := "SrcType := Real" } LE_Contact(in1 := "Moving_Z 1(1)", in2 := 5.0)
      wire#w2
      Coil( "s4(1)" )
   END_RUNG
   RUNG wire#w1
      Contact( "s4(1)" )
   END_RUNG wire#w2
   // the same network as SCL:
   "s4(1)" := "s3(1)" AND (("Moving_Z 1(1)" <= 5.0) OR "s4(1)");
END_REGION

REGION Network 7
   RUNG wire#powerrail
      Contact( "s3(1)" )
      wire#w1
      I_Contact( "s6(1)" )
      Coil( "Grab(1)" )
   END_RUNG
   RUNG wire#powerrail
      Contact( "Grab(1)" )
   END_RUNG wire#w1
   // the same network as SCL:
   "Grab(1)" := ("s3(1)" OR "Grab(1)") AND NOT "s6(1)";
END_REGION

REGION Network 8
   RUNG wire#powerrail
      Contact( "s4(1)" )
      wire#w1
      I_Contact( "s7(1)" )
      Coil( "Move X(1)" )
   END_RUNG
   RUNG wire#powerrail
      Contact( "Move X(1)" )
   END_RUNG wire#w1
   RUNG wire#powerrail
      Contact( "Move X(1)" )
      Move(in := 10.0, out1 => "Move_X 1(1)")
   END_RUNG
   RUNG wire#powerrail
      I_Contact( "Move X(1)" )
      Move(in := 0.0, out1 => "Move_X 1(1)")
   END_RUNG
   // the same network as SCL:
   "Move X(1)" := ("s4(1)" OR "Move X(1)") AND NOT "s7(1)";
   IF "Move X(1)" THEN "Move_X 1(1)" := 10.0; END_IF;
   IF NOT "Move X(1)" THEN "Move_X 1(1)" := 0.0; END_IF;
END_REGION

REGION Network 9
   RUNG wire#powerrail
      Contact( "s4(1)" )
      wire#w1
      { S7_Templates := "SrcType := Real" } GE_Contact(in1 := "Moving_X 1(1)", in2 := 1.0)
      wire#w2
      Coil( "s5(1)" )
   END_RUNG
   RUNG wire#w1
      Contact( "s5(1)" )
   END_RUNG wire#w2
   // the same network as SCL:
   "s5(1)" := "s4(1)" AND (("Moving_X 1(1)" >= 1.0) OR "s5(1)");
END_REGION

REGION Network 10
   RUNG wire#powerrail
      Contact( "s5(1)" )
      wire#w1
      Contact( "Item at Exit(1)" )
      { S7_Templates := "SrcType := Real" } GE_Contact(in1 := "Moving_Z 1(1)", in2 := 5.0)
      wire#w2
      Coil( "s6(1)" )
   END_RUNG
   RUNG wire#w1
      Contact( "s6(1)" )
   END_RUNG wire#w2
   // the same network as SCL:
   "s6(1)" := "s5(1)" AND (("Item at Exit(1)" AND ("Moving_Z 1(1)" >= 5.0)) OR "s6(1)");
END_REGION

REGION Network 11
   RUNG wire#powerrail
      Contact( "s6(1)" )
      wire#w1
      { S7_Templates := "SrcType := Real" } LE_Contact(in1 := "Moving_Z 1(1)", in2 := 5.0)
      wire#w2
      Coil( "s7(1)" )
   END_RUNG
   RUNG wire#w1
      Contact( "s7(1)" )
   END_RUNG wire#w2
   // the same network as SCL:
   "s7(1)" := "s6(1)" AND (("Moving_Z 1(1)" <= 5.0) OR "s7(1)");
END_REGION

REGION Network 12
   RUNG wire#powerrail
      Contact( "s7(1)" )
      wire#w1
      { S7_Templates := "SrcType := Real" } LE_Contact(in1 := "Moving_X 1(1)", in2 := 5.0)
      wire#w2
      Coil( "s8(1)" )
   END_RUNG
   RUNG wire#w1
      Contact( "s8(1)" )
   END_RUNG wire#w2
   // the same network as SCL:
   "s8(1)" := "s7(1)" AND (("Moving_X 1(1)" <= 5.0) OR "s8(1)");
END_REGION

REGION Network 13
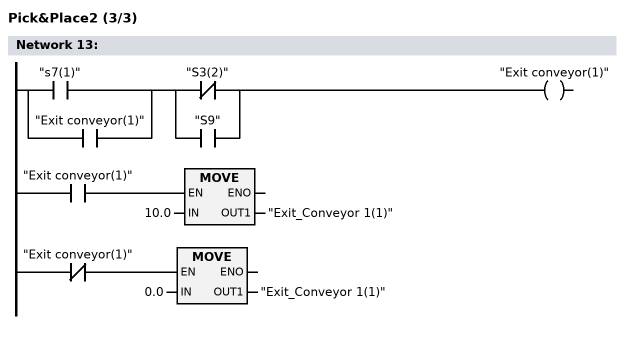
   RUNG wire#powerrail
      Contact( "s7(1)" )
      wire#w1
      I_Contact( "S3(2)" )
      wire#w2
      Coil( "Exit conveyor(1)" )
   END_RUNG
   RUNG wire#powerrail
      Contact( "Exit conveyor(1)" )
   END_RUNG wire#w1
   RUNG wire#w1
      Contact( "S9" )
   END_RUNG wire#w2
   RUNG wire#powerrail
      Contact( "Exit conveyor(1)" )
      Move(in := 10.0, out1 => "Exit_Conveyor 1(1)")
   END_RUNG
   RUNG wire#powerrail
      I_Contact( "Exit conveyor(1)" )
      Move(in := 0.0, out1 => "Exit_Conveyor 1(1)")
   END_RUNG
   // the same network as SCL:
   "Exit conveyor(1)" := ("s7(1)" OR "Exit conveyor(1)") AND (NOT "S3(2)" OR "S9");
   IF "Exit conveyor(1)" THEN "Exit_Conveyor 1(1)" := 10.0; END_IF;
   IF NOT "Exit conveyor(1)" THEN "Exit_Conveyor 1(1)" := 0.0; END_IF;
END_REGION
END_FUNCTION_BLOCK

FUNCTION_BLOCK "machine_center"   // FB3, LAD
{ S7_Optimized_Access := 'TRUE' }
VERSION : 0.1
   VAR_TEMP   // added for the SCL form of the ladder/FBD networks
      _w1 : Bool;
   END_VAR
BEGIN

REGION Network 2: States
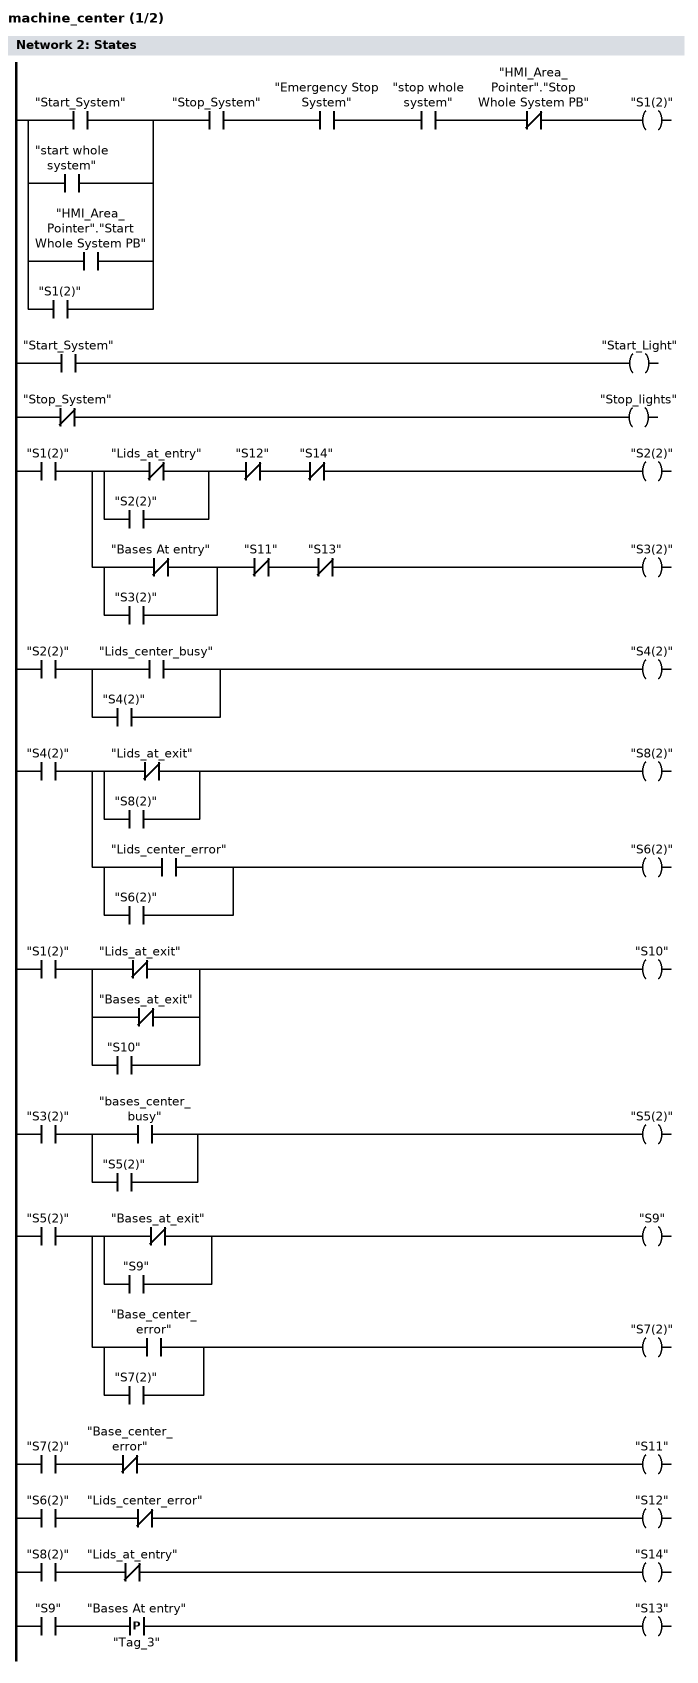
   RUNG wire#powerrail
      Contact( "Start_System" )
      wire#w1
      Contact( "Stop_System" )
      Contact( "Emergency Stop System" )
      Contact( "stop whole system" )
      I_Contact( "HMI_Area_Pointer"."Stop Whole System PB" )
      Coil( "S1(2)" )
   END_RUNG
   RUNG wire#powerrail
      Contact( "start whole system" )
   END_RUNG wire#w1
   RUNG wire#powerrail
      Contact( "HMI_Area_Pointer"."Start Whole System PB" )
   END_RUNG wire#w1
   RUNG wire#powerrail
      Contact( "S1(2)" )
   END_RUNG wire#w1
   RUNG wire#powerrail
      Contact( "Start_System" )
      Coil( "Start_Light" )
   END_RUNG
   RUNG wire#powerrail
      I_Contact( "Stop_System" )
      Coil( "Stop_lights" )
   END_RUNG
   RUNG wire#powerrail
      Contact( "S1(2)" )
      wire#w2
      I_Contact( "Lids_at_entry" )
      wire#w3
      I_Contact( "S12" )
      I_Contact( "S14" )
      Coil( "S2(2)" )
   END_RUNG
   RUNG wire#w2
      Contact( "S2(2)" )
   END_RUNG wire#w3
   RUNG wire#w2
      I_Contact( "Bases At entry" )
      wire#w4
      I_Contact( "S11" )
      I_Contact( "S13" )
      Coil( "S3(2)" )
   END_RUNG
   RUNG wire#w2
      Contact( "S3(2)" )
   END_RUNG wire#w4
   RUNG wire#powerrail
      Contact( "S2(2)" )
      wire#w5
      Contact( "Lids_center_busy" )
      wire#w6
      Coil( "S4(2)" )
   END_RUNG
   RUNG wire#w5
      Contact( "S4(2)" )
   END_RUNG wire#w6
   RUNG wire#powerrail
      Contact( "S4(2)" )
      wire#w7
      I_Contact( "Lids_at_exit" )
      wire#w8
      Coil( "S8(2)" )
   END_RUNG
   RUNG wire#w7
      Contact( "S8(2)" )
   END_RUNG wire#w8
   RUNG wire#w7
      Contact( "Lids_center_error" )
      wire#w9
      Coil( "S6(2)" )
   END_RUNG
   RUNG wire#w7
      Contact( "S6(2)" )
   END_RUNG wire#w9
   RUNG wire#powerrail
      Contact( "S1(2)" )
      wire#w10
      I_Contact( "Lids_at_exit" )
      wire#w11
      Coil( "S10" )
   END_RUNG
   RUNG wire#w10
      I_Contact( "Bases_at_exit" )
   END_RUNG wire#w11
   RUNG wire#w10
      Contact( "S10" )
   END_RUNG wire#w11
   RUNG wire#powerrail
      Contact( "S3(2)" )
      wire#w12
      Contact( "bases_center_busy" )
      wire#w13
      Coil( "S5(2)" )
   END_RUNG
   RUNG wire#w12
      Contact( "S5(2)" )
   END_RUNG wire#w13
   RUNG wire#powerrail
      Contact( "S5(2)" )
      wire#w14
      I_Contact( "Bases_at_exit" )
      wire#w15
      Coil( "S9" )
   END_RUNG
   RUNG wire#w14
      Contact( "S9" )
   END_RUNG wire#w15
   RUNG wire#w14
      Contact( "Base_center_error" )
      wire#w16
      Coil( "S7(2)" )
   END_RUNG
   RUNG wire#w14
      Contact( "S7(2)" )
   END_RUNG wire#w16
   RUNG wire#powerrail
      Contact( "S7(2)" )
      I_Contact( "Base_center_error" )
      Coil( "S11" )
   END_RUNG
   RUNG wire#powerrail
      Contact( "S6(2)" )
      I_Contact( "Lids_center_error" )
      Coil( "S12" )
   END_RUNG
   RUNG wire#powerrail
      Contact( "S8(2)" )
      I_Contact( "Lids_at_entry" )
      Coil( "S14" )
   END_RUNG
   RUNG wire#powerrail
      Contact( "S9" )
      P_Contact(operand := "Bases At entry", bit := "Tag_3")
      Coil( "S13" )
   END_RUNG
   // the same network as SCL:
   "S1(2)" := ("Start_System" OR "start whole system" OR "HMI_Area_Pointer"."Start Whole System PB" OR "S1(2)") AND "Stop_System" AND "Emergency Stop System" AND "stop whole system" AND NOT "HMI_Area_Pointer"."Stop Whole System PB";
   "Start_Light" := "Start_System";
   "Stop_lights" := NOT "Stop_System";
   "S2(2)" := "S1(2)" AND (NOT "Lids_at_entry" OR "S2(2)") AND NOT "S12" AND NOT "S14";
   "S3(2)" := "S1(2)" AND (NOT "Bases At entry" OR "S3(2)") AND NOT "S11" AND NOT "S13";
   "S4(2)" := "S2(2)" AND ("Lids_center_busy" OR "S4(2)");
   "S8(2)" := "S4(2)" AND (NOT "Lids_at_exit" OR "S8(2)");
   "S6(2)" := "S4(2)" AND ("Lids_center_error" OR "S6(2)");
   "S10" := "S1(2)" AND (NOT "Lids_at_exit" OR NOT "Bases_at_exit" OR "S10");
   "S5(2)" := "S3(2)" AND ("bases_center_busy" OR "S5(2)");
   "S9" := "S5(2)" AND (NOT "Bases_at_exit" OR "S9");
   "S7(2)" := "S5(2)" AND ("Base_center_error" OR "S7(2)");
   "S11" := "S7(2)" AND NOT "Base_center_error";
   "S12" := "S6(2)" AND NOT "Lids_center_error";
   "S14" := "S8(2)" AND NOT "Lids_at_entry";
   #_w1 := "S9" AND "Bases At entry" AND NOT "Tag_3";   // rising edge of "Bases At entry"
   "Tag_3" := "Bases At entry";
   "S13" := #_w1;
END_REGION

REGION Network 3: ACTUATORS
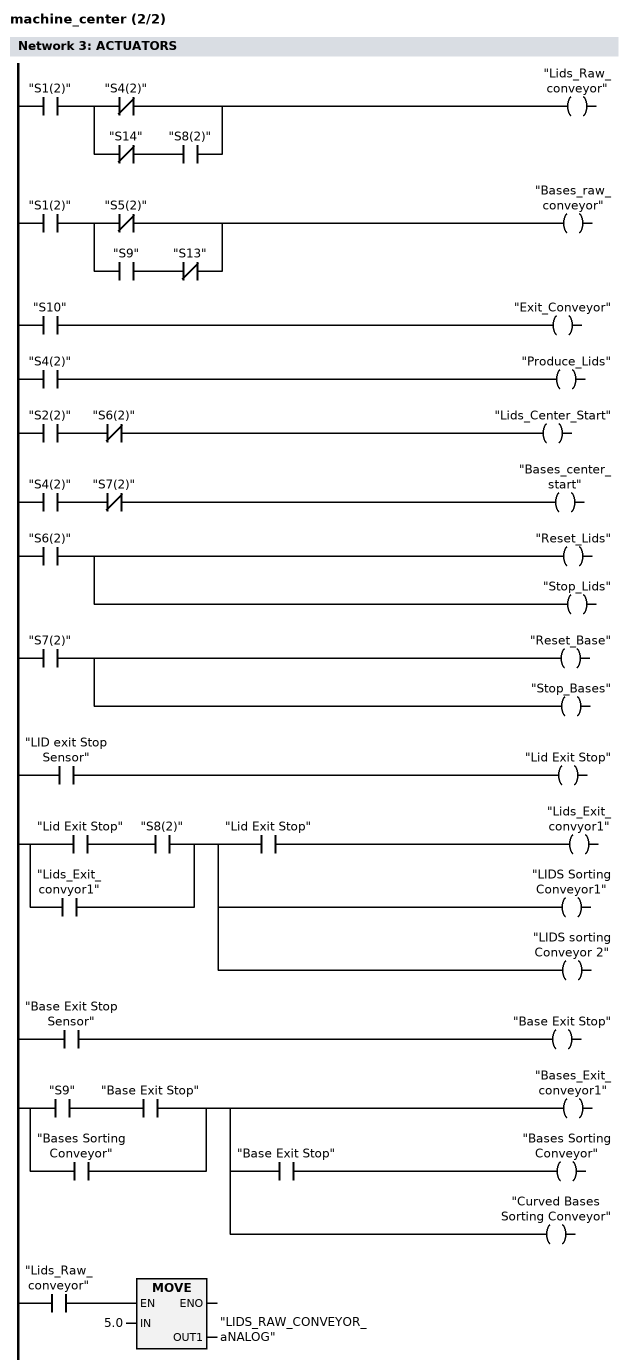
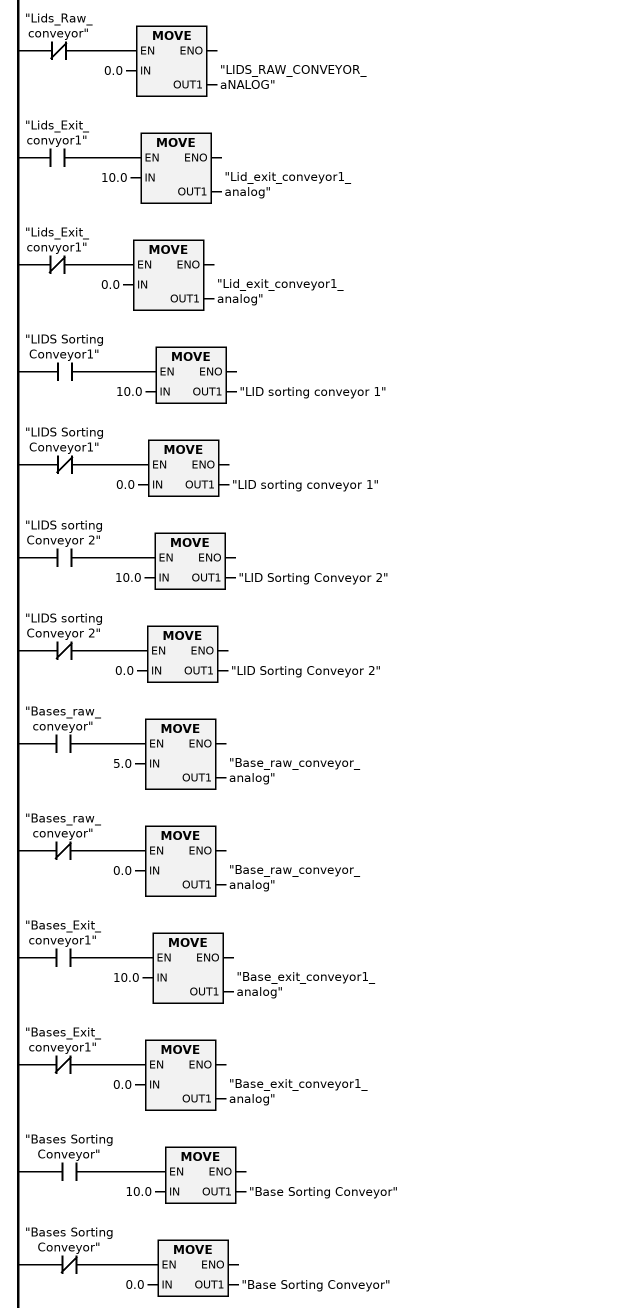
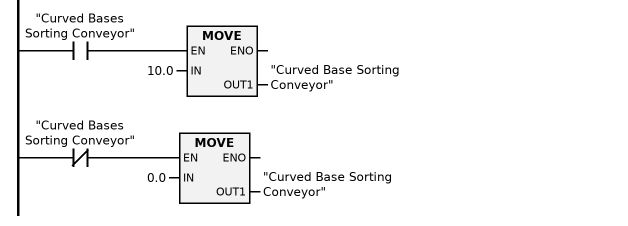
   RUNG wire#powerrail
      Contact( "S1(2)" )
      wire#w1
      I_Contact( "S4(2)" )
      wire#w2
      Coil( "Lids_Raw_conveyor" )
   END_RUNG
   RUNG wire#w1
      I_Contact( "S14" )
      Contact( "S8(2)" )
   END_RUNG wire#w2
   RUNG wire#powerrail
      Contact( "S1(2)" )
      wire#w3
      I_Contact( "S5(2)" )
      wire#w4
      Coil( "Bases_raw_conveyor" )
   END_RUNG
   RUNG wire#w3
      Contact( "S9" )
      I_Contact( "S13" )
   END_RUNG wire#w4
   RUNG wire#powerrail
      Contact( "S10" )
      Coil( "Exit_Conveyor" )
   END_RUNG
   RUNG wire#powerrail
      Contact( "S4(2)" )
      Coil( "Produce_Lids" )
   END_RUNG
   RUNG wire#powerrail
      Contact( "S2(2)" )
      I_Contact( "S6(2)" )
      Coil( "Lids_Center_Start" )
   END_RUNG
   RUNG wire#powerrail
      Contact( "S4(2)" )
      I_Contact( "S7(2)" )
      Coil( "Bases_center_start" )
   END_RUNG
   RUNG wire#powerrail
      Contact( "S6(2)" )
      wire#w5
      Coil( "Reset_Lids" )
   END_RUNG
   RUNG wire#w5
      Coil( "Stop_Lids" )
   END_RUNG
   RUNG wire#powerrail
      Contact( "S7(2)" )
      wire#w6
      Coil( "Reset_Base" )
   END_RUNG
   RUNG wire#w6
      Coil( "Stop_Bases" )
   END_RUNG
   RUNG wire#powerrail
      Contact( "LID exit Stop Sensor" )
      Coil( "Lid Exit Stop" )
   END_RUNG
   RUNG wire#powerrail
      Contact( "Lid Exit Stop" )
      Contact( "S8(2)" )
      wire#w7
      Contact( "Lid Exit Stop" )
      Coil( "Lids_Exit_convyor1" )
   END_RUNG
   RUNG wire#powerrail
      Contact( "Lids_Exit_convyor1" )
   END_RUNG wire#w7
   RUNG wire#w7
      Coil( "LIDS Sorting Conveyor1" )
   END_RUNG
   RUNG wire#w7
      Coil( "LIDS sorting Conveyor 2" )
   END_RUNG
   RUNG wire#powerrail
      Contact( "Base Exit Stop Sensor" )
      Coil( "Base Exit Stop" )
   END_RUNG
   RUNG wire#powerrail
      Contact( "S9" )
      Contact( "Base Exit Stop" )
      wire#w8
      Coil( "Bases_Exit_conveyor1" )
   END_RUNG
   RUNG wire#powerrail
      Contact( "Bases Sorting Conveyor" )
   END_RUNG wire#w8
   RUNG wire#w8
      Contact( "Base Exit Stop" )
      Coil( "Bases Sorting Conveyor" )
   END_RUNG
   RUNG wire#w8
      Coil( "Curved Bases Sorting Conveyor" )
   END_RUNG
   RUNG wire#powerrail
      Contact( "Lids_Raw_conveyor" )
      Move(in := 5.0, out1 => "LIDS_RAW_CONVEYOR_aNALOG")
   END_RUNG
   RUNG wire#powerrail
      I_Contact( "Lids_Raw_conveyor" )
      Move(in := 0.0, out1 => "LIDS_RAW_CONVEYOR_aNALOG")
   END_RUNG
   RUNG wire#powerrail
      Contact( "Lids_Exit_convyor1" )
      Move(in := 10.0, out1 => "Lid_exit_conveyor1_analog")
   END_RUNG
   RUNG wire#powerrail
      I_Contact( "Lids_Exit_convyor1" )
      Move(in := 0.0, out1 => "Lid_exit_conveyor1_analog")
   END_RUNG
   RUNG wire#powerrail
      Contact( "LIDS Sorting Conveyor1" )
      Move(in := 10.0, out1 => "LID sorting conveyor 1")
   END_RUNG
   RUNG wire#powerrail
      I_Contact( "LIDS Sorting Conveyor1" )
      Move(in := 0.0, out1 => "LID sorting conveyor 1")
   END_RUNG
   RUNG wire#powerrail
      Contact( "LIDS sorting Conveyor 2" )
      Move(in := 10.0, out1 => "LID Sorting Conveyor 2")
   END_RUNG
   RUNG wire#powerrail
      I_Contact( "LIDS sorting Conveyor 2" )
      Move(in := 0.0, out1 => "LID Sorting Conveyor 2")
   END_RUNG
   RUNG wire#powerrail
      Contact( "Bases_raw_conveyor" )
      Move(in := 5.0, out1 => "Base_raw_conveyor_analog")
   END_RUNG
   RUNG wire#powerrail
      I_Contact( "Bases_raw_conveyor" )
      Move(in := 0.0, out1 => "Base_raw_conveyor_analog")
   END_RUNG
   RUNG wire#powerrail
      Contact( "Bases_Exit_conveyor1" )
      Move(in := 10.0, out1 => "Base_exit_conveyor1_analog")
   END_RUNG
   RUNG wire#powerrail
      I_Contact( "Bases_Exit_conveyor1" )
      Move(in := 0.0, out1 => "Base_exit_conveyor1_analog")
   END_RUNG
   RUNG wire#powerrail
      Contact( "Bases Sorting Conveyor" )
      Move(in := 10.0, out1 => "Base Sorting Conveyor")
   END_RUNG
   RUNG wire#powerrail
      I_Contact( "Bases Sorting Conveyor" )
      Move(in := 0.0, out1 => "Base Sorting Conveyor")
   END_RUNG
   RUNG wire#powerrail
      Contact( "Curved Bases Sorting Conveyor" )
      Move(in := 10.0, out1 => "Curved Base Sorting Conveyor")
   END_RUNG
   RUNG wire#powerrail
      I_Contact( "Curved Bases Sorting Conveyor" )
      Move(in := 0.0, out1 => "Curved Base Sorting Conveyor")
   END_RUNG
   // the same network as SCL:
   "Lids_Raw_conveyor" := "S1(2)" AND (NOT "S4(2)" OR (NOT "S14" AND "S8(2)"));
   "Bases_raw_conveyor" := "S1(2)" AND (NOT "S5(2)" OR ("S9" AND NOT "S13"));
   "Exit_Conveyor" := "S10";
   "Produce_Lids" := "S4(2)";
   "Lids_Center_Start" := "S2(2)" AND NOT "S6(2)";
   "Bases_center_start" := "S4(2)" AND NOT "S7(2)";
   "Reset_Lids" := "S6(2)";
   "Stop_Lids" := "S6(2)";
   "Reset_Base" := "S7(2)";
   "Stop_Bases" := "S7(2)";
   "Lid Exit Stop" := "LID exit Stop Sensor";
   #_w1 := ("Lid Exit Stop" AND "S8(2)") OR "Lids_Exit_convyor1";
   "Lids_Exit_convyor1" := #_w1 AND "Lid Exit Stop";
   "LIDS Sorting Conveyor1" := #_w1;
   "LIDS sorting Conveyor 2" := #_w1;
   "Base Exit Stop" := "Base Exit Stop Sensor";
   "Bases_Exit_conveyor1" := ("S9" AND "Base Exit Stop") OR "Bases Sorting Conveyor";
   "Bases Sorting Conveyor" := "Bases_Exit_conveyor1" AND "Base Exit Stop";
   "Curved Bases Sorting Conveyor" := "Bases_Exit_conveyor1";
   IF "Lids_Raw_conveyor" THEN "LIDS_RAW_CONVEYOR_aNALOG" := 5.0; END_IF;
   IF NOT "Lids_Raw_conveyor" THEN "LIDS_RAW_CONVEYOR_aNALOG" := 0.0; END_IF;
   IF "Lids_Exit_convyor1" THEN "Lid_exit_conveyor1_analog" := 10.0; END_IF;
   IF NOT "Lids_Exit_convyor1" THEN "Lid_exit_conveyor1_analog" := 0.0; END_IF;
   IF "LIDS Sorting Conveyor1" THEN "LID sorting conveyor 1" := 10.0; END_IF;
   IF NOT "LIDS Sorting Conveyor1" THEN "LID sorting conveyor 1" := 0.0; END_IF;
   IF "LIDS sorting Conveyor 2" THEN "LID Sorting Conveyor 2" := 10.0; END_IF;
   IF NOT "LIDS sorting Conveyor 2" THEN "LID Sorting Conveyor 2" := 0.0; END_IF;
   IF "Bases_raw_conveyor" THEN "Base_raw_conveyor_analog" := 5.0; END_IF;
   IF NOT "Bases_raw_conveyor" THEN "Base_raw_conveyor_analog" := 0.0; END_IF;
   IF "Bases_Exit_conveyor1" THEN "Base_exit_conveyor1_analog" := 10.0; END_IF;
   IF NOT "Bases_Exit_conveyor1" THEN "Base_exit_conveyor1_analog" := 0.0; END_IF;
   IF "Bases Sorting Conveyor" THEN "Base Sorting Conveyor" := 10.0; END_IF;
   IF NOT "Bases Sorting Conveyor" THEN "Base Sorting Conveyor" := 0.0; END_IF;
   IF "Curved Bases Sorting Conveyor" THEN "Curved Base Sorting Conveyor" := 10.0; END_IF;
   IF NOT "Curved Bases Sorting Conveyor" THEN "Curved Base Sorting Conveyor" := 0.0; END_IF;
END_REGION
END_FUNCTION_BLOCK

FUNCTION_BLOCK "Sorting1"   // FB4, LAD
{ S7_Optimized_Access := 'TRUE' }
VERSION : 0.1
BEGIN

REGION Network 1
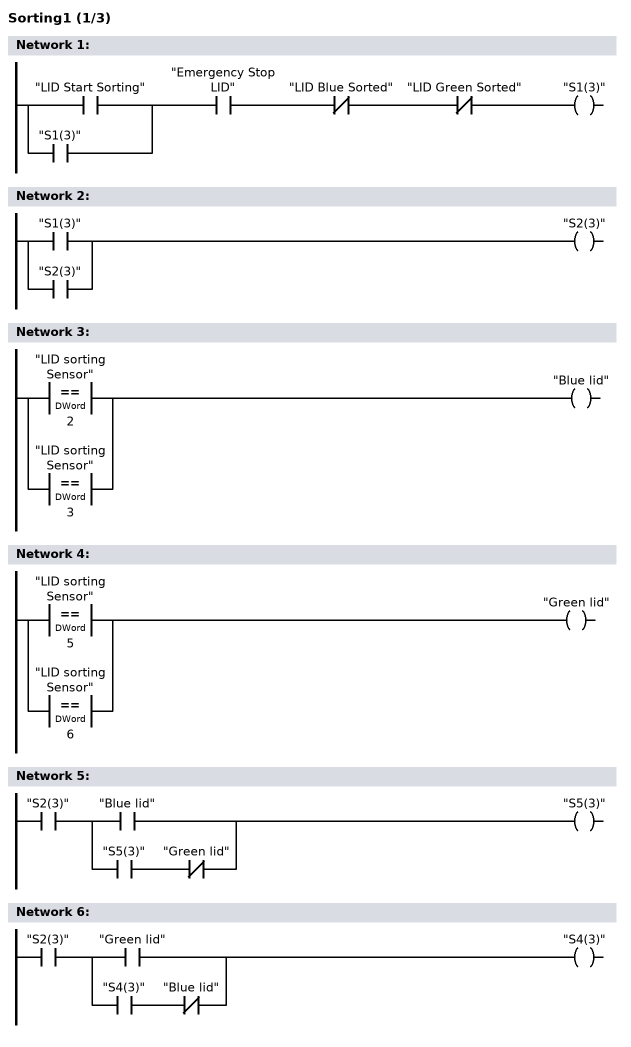
   RUNG wire#powerrail
      Contact( "LID Start Sorting" )
      wire#w1
      Contact( "Emergency Stop LID" )
      I_Contact( "LID Blue Sorted" )
      I_Contact( "LID Green Sorted" )
      Coil( "S1(3)" )
   END_RUNG
   RUNG wire#powerrail
      Contact( "S1(3)" )
   END_RUNG wire#w1
   // the same network as SCL:
   "S1(3)" := ("LID Start Sorting" OR "S1(3)") AND "Emergency Stop LID" AND NOT "LID Blue Sorted" AND NOT "LID Green Sorted";
END_REGION

REGION Network 2
   RUNG wire#powerrail
      Contact( "S1(3)" )
      wire#w1
      Coil( "S2(3)" )
   END_RUNG
   RUNG wire#powerrail
      Contact( "S2(3)" )
   END_RUNG wire#w1
   // the same network as SCL:
   "S2(3)" := "S1(3)" OR "S2(3)";
END_REGION

REGION Network 3
   RUNG wire#powerrail
      { S7_Templates := "SrcType := DWord" } EQ_Contact(in1 := "LID sorting Sensor", in2 := 2)
      wire#w1
      Coil( "Blue lid" )
   END_RUNG
   RUNG wire#powerrail
      { S7_Templates := "SrcType := DWord" } EQ_Contact(in1 := "LID sorting Sensor", in2 := 3)
   END_RUNG wire#w1
   // the same network as SCL:
   "Blue lid" := ("LID sorting Sensor" = 2) OR ("LID sorting Sensor" = 3);
END_REGION

REGION Network 4
   RUNG wire#powerrail
      { S7_Templates := "SrcType := DWord" } EQ_Contact(in1 := "LID sorting Sensor", in2 := 5)
      wire#w1
      Coil( "Green lid" )
   END_RUNG
   RUNG wire#powerrail
      { S7_Templates := "SrcType := DWord" } EQ_Contact(in1 := "LID sorting Sensor", in2 := 6)
   END_RUNG wire#w1
   // the same network as SCL:
   "Green lid" := ("LID sorting Sensor" = 5) OR ("LID sorting Sensor" = 6);
END_REGION

REGION Network 5
   RUNG wire#powerrail
      Contact( "S2(3)" )
      wire#w1
      Contact( "Blue lid" )
      wire#w2
      Coil( "S5(3)" )
   END_RUNG
   RUNG wire#w1
      Contact( "S5(3)" )
      I_Contact( "Green lid" )
   END_RUNG wire#w2
   // the same network as SCL:
   "S5(3)" := "S2(3)" AND ("Blue lid" OR ("S5(3)" AND NOT "Green lid"));
END_REGION

REGION Network 6
   RUNG wire#powerrail
      Contact( "S2(3)" )
      wire#w1
      Contact( "Green lid" )
      wire#w2
      Coil( "S4(3)" )
   END_RUNG
   RUNG wire#w1
      Contact( "S4(3)" )
      I_Contact( "Blue lid" )
   END_RUNG wire#w2
   // the same network as SCL:
   "S4(3)" := "S2(3)" AND ("Green lid" OR ("S4(3)" AND NOT "Blue lid"));
END_REGION

REGION Network 7
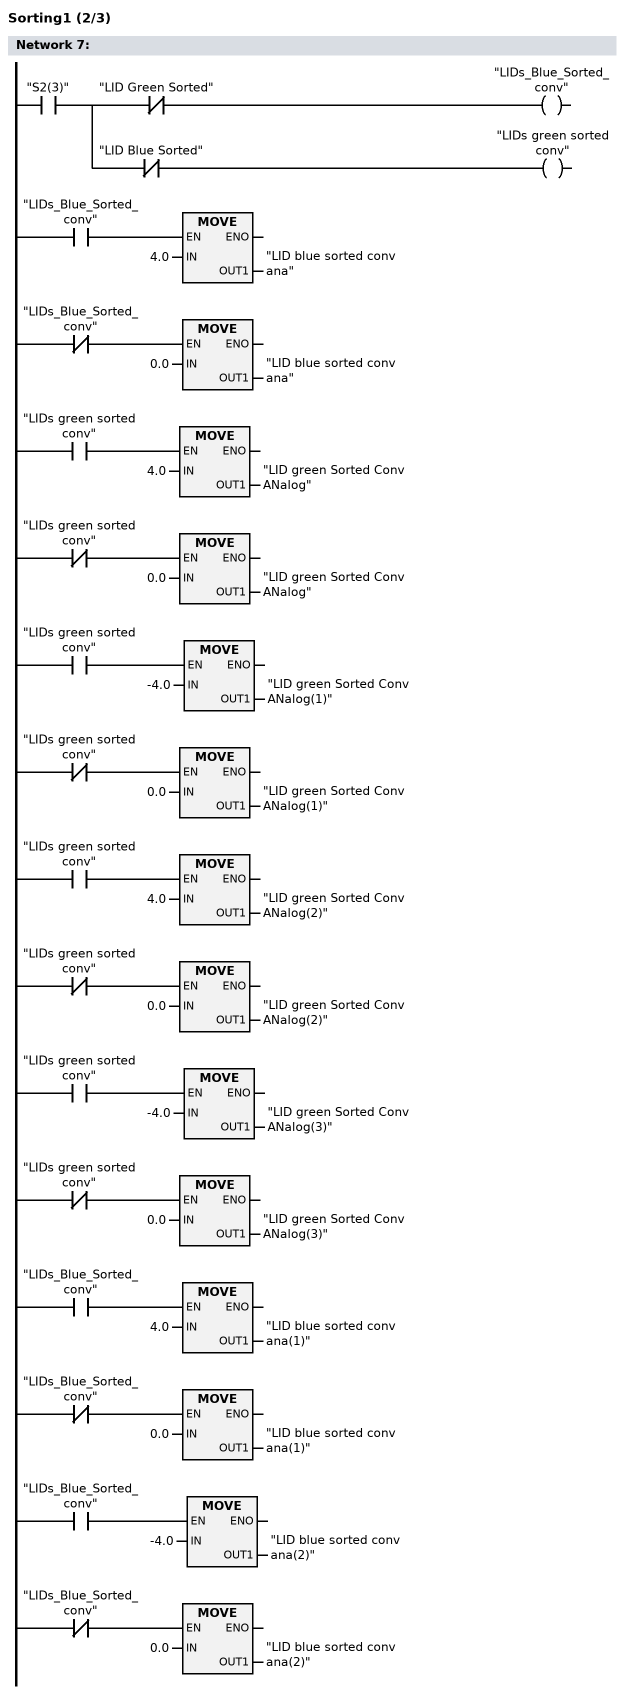
   RUNG wire#powerrail
      Contact( "S2(3)" )
      wire#w1
      I_Contact( "LID Green Sorted" )
      Coil( "LIDs_Blue_Sorted_conv" )
   END_RUNG
   RUNG wire#w1
      I_Contact( "LID Blue Sorted" )
      Coil( "LIDs green sorted conv" )
   END_RUNG
   RUNG wire#powerrail
      Contact( "LIDs_Blue_Sorted_conv" )
      Move(in := 4.0, out1 => "LID blue sorted conv ana")
   END_RUNG
   RUNG wire#powerrail
      I_Contact( "LIDs_Blue_Sorted_conv" )
      Move(in := 0.0, out1 => "LID blue sorted conv ana")
   END_RUNG
   RUNG wire#powerrail
      Contact( "LIDs green sorted conv" )
      Move(in := 4.0, out1 => "LID green Sorted Conv ANalog")
   END_RUNG
   RUNG wire#powerrail
      I_Contact( "LIDs green sorted conv" )
      Move(in := 0.0, out1 => "LID green Sorted Conv ANalog")
   END_RUNG
   RUNG wire#powerrail
      Contact( "LIDs green sorted conv" )
      Move(in := -4.0, out1 => "LID green Sorted Conv ANalog(1)")
   END_RUNG
   RUNG wire#powerrail
      I_Contact( "LIDs green sorted conv" )
      Move(in := 0.0, out1 => "LID green Sorted Conv ANalog(1)")
   END_RUNG
   RUNG wire#powerrail
      Contact( "LIDs green sorted conv" )
      Move(in := 4.0, out1 => "LID green Sorted Conv ANalog(2)")
   END_RUNG
   RUNG wire#powerrail
      I_Contact( "LIDs green sorted conv" )
      Move(in := 0.0, out1 => "LID green Sorted Conv ANalog(2)")
   END_RUNG
   RUNG wire#powerrail
      Contact( "LIDs green sorted conv" )
      Move(in := -4.0, out1 => "LID green Sorted Conv ANalog(3)")
   END_RUNG
   RUNG wire#powerrail
      I_Contact( "LIDs green sorted conv" )
      Move(in := 0.0, out1 => "LID green Sorted Conv ANalog(3)")
   END_RUNG
   RUNG wire#powerrail
      Contact( "LIDs_Blue_Sorted_conv" )
      Move(in := 4.0, out1 => "LID blue sorted conv ana(1)")
   END_RUNG
   RUNG wire#powerrail
      I_Contact( "LIDs_Blue_Sorted_conv" )
      Move(in := 0.0, out1 => "LID blue sorted conv ana(1)")
   END_RUNG
   RUNG wire#powerrail
      Contact( "LIDs_Blue_Sorted_conv" )
      Move(in := -4.0, out1 => "LID blue sorted conv ana(2)")
   END_RUNG
   RUNG wire#powerrail
      I_Contact( "LIDs_Blue_Sorted_conv" )
      Move(in := 0.0, out1 => "LID blue sorted conv ana(2)")
   END_RUNG
   // the same network as SCL:
   "LIDs_Blue_Sorted_conv" := "S2(3)" AND NOT "LID Green Sorted";
   "LIDs green sorted conv" := "S2(3)" AND NOT "LID Blue Sorted";
   IF "LIDs_Blue_Sorted_conv" THEN "LID blue sorted conv ana" := 4.0; END_IF;
   IF NOT "LIDs_Blue_Sorted_conv" THEN "LID blue sorted conv ana" := 0.0; END_IF;
   IF "LIDs green sorted conv" THEN "LID green Sorted Conv ANalog" := 4.0; END_IF;
   IF NOT "LIDs green sorted conv" THEN "LID green Sorted Conv ANalog" := 0.0; END_IF;
   IF "LIDs green sorted conv" THEN "LID green Sorted Conv ANalog(1)" := -4.0; END_IF;
   IF NOT "LIDs green sorted conv" THEN "LID green Sorted Conv ANalog(1)" := 0.0; END_IF;
   IF "LIDs green sorted conv" THEN "LID green Sorted Conv ANalog(2)" := 4.0; END_IF;
   IF NOT "LIDs green sorted conv" THEN "LID green Sorted Conv ANalog(2)" := 0.0; END_IF;
   IF "LIDs green sorted conv" THEN "LID green Sorted Conv ANalog(3)" := -4.0; END_IF;
   IF NOT "LIDs green sorted conv" THEN "LID green Sorted Conv ANalog(3)" := 0.0; END_IF;
   IF "LIDs_Blue_Sorted_conv" THEN "LID blue sorted conv ana(1)" := 4.0; END_IF;
   IF NOT "LIDs_Blue_Sorted_conv" THEN "LID blue sorted conv ana(1)" := 0.0; END_IF;
   IF "LIDs_Blue_Sorted_conv" THEN "LID blue sorted conv ana(2)" := -4.0; END_IF;
   IF NOT "LIDs_Blue_Sorted_conv" THEN "LID blue sorted conv ana(2)" := 0.0; END_IF;
END_REGION

REGION Network 8
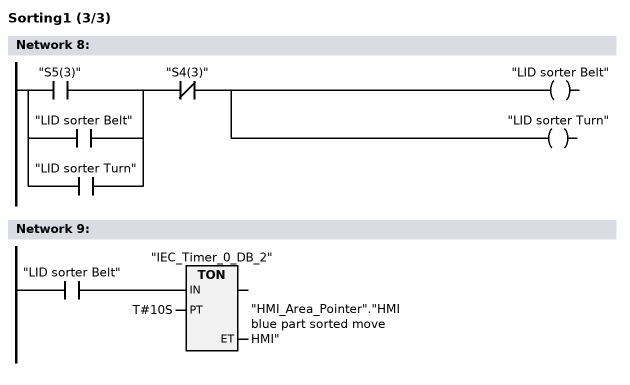
   RUNG wire#powerrail
      Contact( "S5(3)" )
      wire#w1
      I_Contact( "S4(3)" )
      wire#w2
      Coil( "LID sorter Belt" )
   END_RUNG
   RUNG wire#powerrail
      Contact( "LID sorter Belt" )
   END_RUNG wire#w1
   RUNG wire#powerrail
      Contact( "LID sorter Turn" )
   END_RUNG wire#w1
   RUNG wire#w2
      Coil( "LID sorter Turn" )
   END_RUNG
   // the same network as SCL:
   "LID sorter Belt" := ("S5(3)" OR "LID sorter Belt" OR "LID sorter Turn") AND NOT "S4(3)";
   "LID sorter Turn" := "LID sorter Belt";
END_REGION

REGION Network 9
   "IEC_Timer_0_DB_2".TON(IN := "LID sorter Belt",
                          PT := T#10S,
                          ET => "HMI_Area_Pointer"."HMI blue part sorted move HMI");
END_REGION
END_FUNCTION_BLOCK

FUNCTION_BLOCK "Sorting2"   // FB5, LAD
{ S7_Optimized_Access := 'TRUE' }
VERSION : 0.1
BEGIN

REGION Network 1
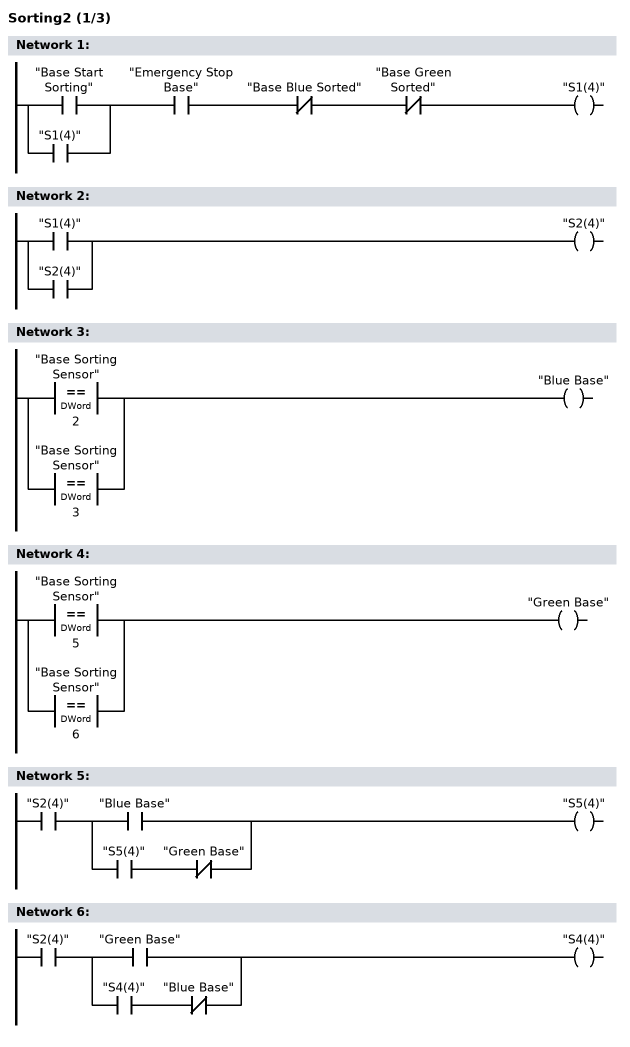
   RUNG wire#powerrail
      Contact( "Base Start Sorting" )
      wire#w1
      Contact( "Emergency Stop Base" )
      I_Contact( "Base Blue Sorted" )
      I_Contact( "Base Green Sorted" )
      Coil( "S1(4)" )
   END_RUNG
   RUNG wire#powerrail
      Contact( "S1(4)" )
   END_RUNG wire#w1
   // the same network as SCL:
   "S1(4)" := ("Base Start Sorting" OR "S1(4)") AND "Emergency Stop Base" AND NOT "Base Blue Sorted" AND NOT "Base Green Sorted";
END_REGION

REGION Network 2
   RUNG wire#powerrail
      Contact( "S1(4)" )
      wire#w1
      Coil( "S2(4)" )
   END_RUNG
   RUNG wire#powerrail
      Contact( "S2(4)" )
   END_RUNG wire#w1
   // the same network as SCL:
   "S2(4)" := "S1(4)" OR "S2(4)";
END_REGION

REGION Network 3
   RUNG wire#powerrail
      { S7_Templates := "SrcType := DWord" } EQ_Contact(in1 := "Base Sorting Sensor", in2 := 2)
      wire#w1
      Coil( "Blue Base" )
   END_RUNG
   RUNG wire#powerrail
      { S7_Templates := "SrcType := DWord" } EQ_Contact(in1 := "Base Sorting Sensor", in2 := 3)
   END_RUNG wire#w1
   // the same network as SCL:
   "Blue Base" := ("Base Sorting Sensor" = 2) OR ("Base Sorting Sensor" = 3);
END_REGION

REGION Network 4
   RUNG wire#powerrail
      { S7_Templates := "SrcType := DWord" } EQ_Contact(in1 := "Base Sorting Sensor", in2 := 5)
      wire#w1
      Coil( "Green Base" )
   END_RUNG
   RUNG wire#powerrail
      { S7_Templates := "SrcType := DWord" } EQ_Contact(in1 := "Base Sorting Sensor", in2 := 6)
   END_RUNG wire#w1
   // the same network as SCL:
   "Green Base" := ("Base Sorting Sensor" = 5) OR ("Base Sorting Sensor" = 6);
END_REGION

REGION Network 5
   RUNG wire#powerrail
      Contact( "S2(4)" )
      wire#w1
      Contact( "Blue Base" )
      wire#w2
      Coil( "S5(4)" )
   END_RUNG
   RUNG wire#w1
      Contact( "S5(4)" )
      I_Contact( "Green Base" )
   END_RUNG wire#w2
   // the same network as SCL:
   "S5(4)" := "S2(4)" AND ("Blue Base" OR ("S5(4)" AND NOT "Green Base"));
END_REGION

REGION Network 6
   RUNG wire#powerrail
      Contact( "S2(4)" )
      wire#w1
      Contact( "Green Base" )
      wire#w2
      Coil( "S4(4)" )
   END_RUNG
   RUNG wire#w1
      Contact( "S4(4)" )
      I_Contact( "Blue Base" )
   END_RUNG wire#w2
   // the same network as SCL:
   "S4(4)" := "S2(4)" AND ("Green Base" OR ("S4(4)" AND NOT "Blue Base"));
END_REGION

REGION Network 7
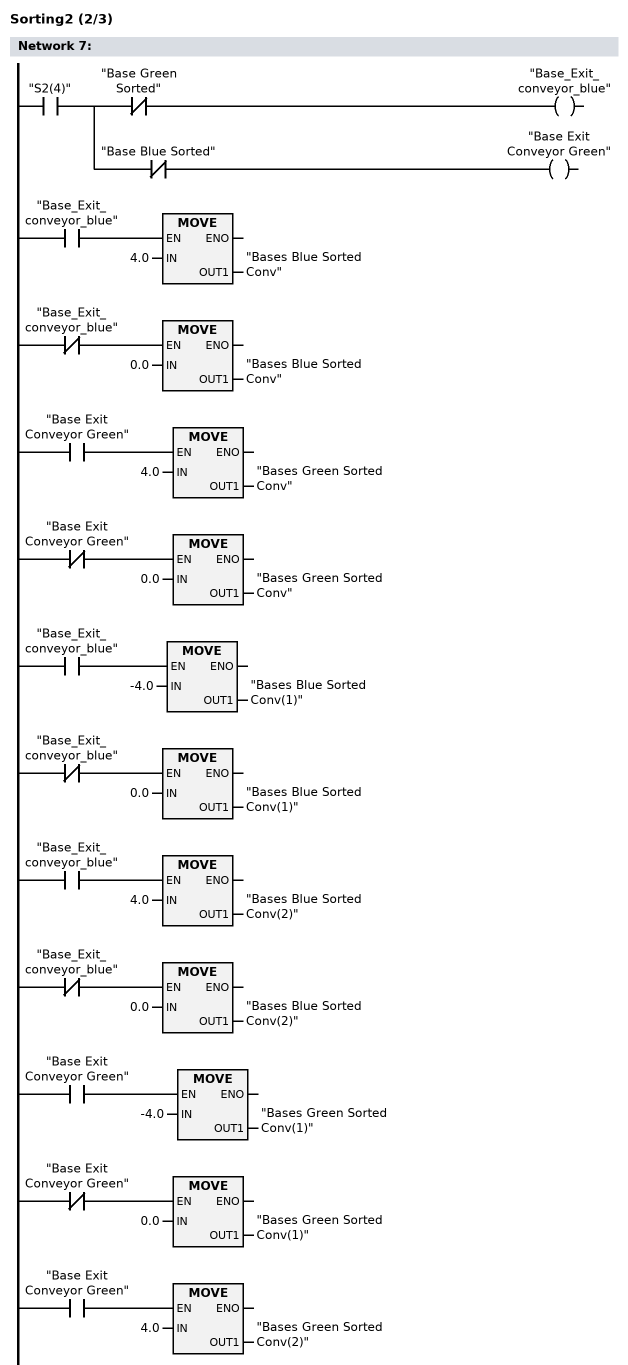
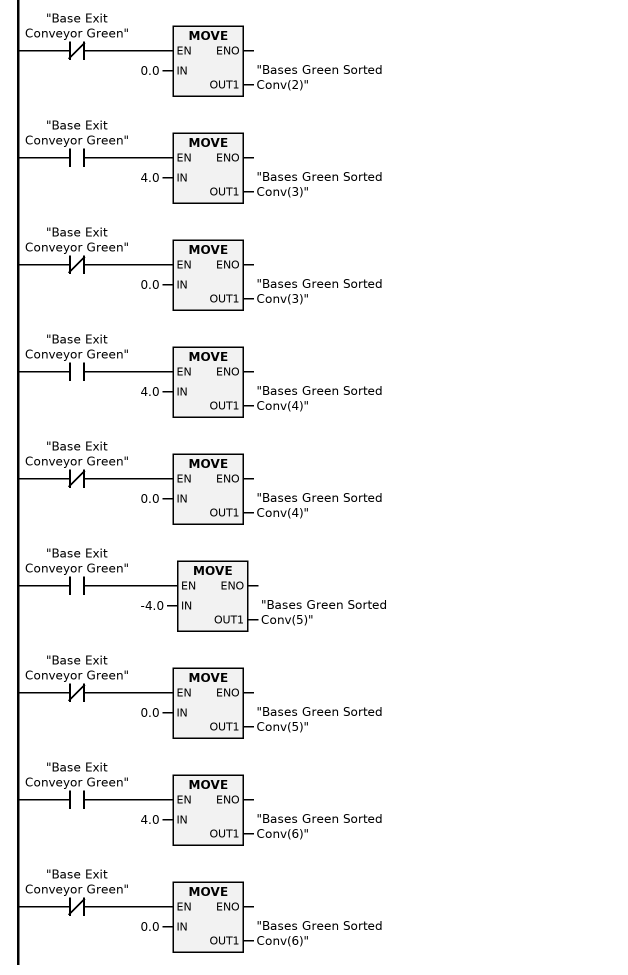
   RUNG wire#powerrail
      Contact( "S2(4)" )
      wire#w1
      I_Contact( "Base Green Sorted" )
      Coil( "Base_Exit_conveyor_blue" )
   END_RUNG
   RUNG wire#w1
      I_Contact( "Base Blue Sorted" )
      Coil( "Base Exit Conveyor Green" )
   END_RUNG
   RUNG wire#powerrail
      Contact( "Base_Exit_conveyor_blue" )
      Move(in := 4.0, out1 => "Bases Blue Sorted Conv")
   END_RUNG
   RUNG wire#powerrail
      I_Contact( "Base_Exit_conveyor_blue" )
      Move(in := 0.0, out1 => "Bases Blue Sorted Conv")
   END_RUNG
   RUNG wire#powerrail
      Contact( "Base Exit Conveyor Green" )
      Move(in := 4.0, out1 => "Bases Green Sorted Conv")
   END_RUNG
   RUNG wire#powerrail
      I_Contact( "Base Exit Conveyor Green" )
      Move(in := 0.0, out1 => "Bases Green Sorted Conv")
   END_RUNG
   RUNG wire#powerrail
      Contact( "Base_Exit_conveyor_blue" )
      Move(in := -4.0, out1 => "Bases Blue Sorted Conv(1)")
   END_RUNG
   RUNG wire#powerrail
      I_Contact( "Base_Exit_conveyor_blue" )
      Move(in := 0.0, out1 => "Bases Blue Sorted Conv(1)")
   END_RUNG
   RUNG wire#powerrail
      Contact( "Base_Exit_conveyor_blue" )
      Move(in := 4.0, out1 => "Bases Blue Sorted Conv(2)")
   END_RUNG
   RUNG wire#powerrail
      I_Contact( "Base_Exit_conveyor_blue" )
      Move(in := 0.0, out1 => "Bases Blue Sorted Conv(2)")
   END_RUNG
   RUNG wire#powerrail
      Contact( "Base Exit Conveyor Green" )
      Move(in := -4.0, out1 => "Bases Green Sorted Conv(1)")
   END_RUNG
   RUNG wire#powerrail
      I_Contact( "Base Exit Conveyor Green" )
      Move(in := 0.0, out1 => "Bases Green Sorted Conv(1)")
   END_RUNG
   RUNG wire#powerrail
      Contact( "Base Exit Conveyor Green" )
      Move(in := 4.0, out1 => "Bases Green Sorted Conv(2)")
   END_RUNG
   RUNG wire#powerrail
      I_Contact( "Base Exit Conveyor Green" )
      Move(in := 0.0, out1 => "Bases Green Sorted Conv(2)")
   END_RUNG
   RUNG wire#powerrail
      Contact( "Base Exit Conveyor Green" )
      Move(in := 4.0, out1 => "Bases Green Sorted Conv(3)")
   END_RUNG
   RUNG wire#powerrail
      I_Contact( "Base Exit Conveyor Green" )
      Move(in := 0.0, out1 => "Bases Green Sorted Conv(3)")
   END_RUNG
   RUNG wire#powerrail
      Contact( "Base Exit Conveyor Green" )
      Move(in := 4.0, out1 => "Bases Green Sorted Conv(4)")
   END_RUNG
   RUNG wire#powerrail
      I_Contact( "Base Exit Conveyor Green" )
      Move(in := 0.0, out1 => "Bases Green Sorted Conv(4)")
   END_RUNG
   RUNG wire#powerrail
      Contact( "Base Exit Conveyor Green" )
      Move(in := -4.0, out1 => "Bases Green Sorted Conv(5)")
   END_RUNG
   RUNG wire#powerrail
      I_Contact( "Base Exit Conveyor Green" )
      Move(in := 0.0, out1 => "Bases Green Sorted Conv(5)")
   END_RUNG
   RUNG wire#powerrail
      Contact( "Base Exit Conveyor Green" )
      Move(in := 4.0, out1 => "Bases Green Sorted Conv(6)")
   END_RUNG
   RUNG wire#powerrail
      I_Contact( "Base Exit Conveyor Green" )
      Move(in := 0.0, out1 => "Bases Green Sorted Conv(6)")
   END_RUNG
   // the same network as SCL:
   "Base_Exit_conveyor_blue" := "S2(4)" AND NOT "Base Green Sorted";
   "Base Exit Conveyor Green" := "S2(4)" AND NOT "Base Blue Sorted";
   IF "Base_Exit_conveyor_blue" THEN "Bases Blue Sorted Conv" := 4.0; END_IF;
   IF NOT "Base_Exit_conveyor_blue" THEN "Bases Blue Sorted Conv" := 0.0; END_IF;
   IF "Base Exit Conveyor Green" THEN "Bases Green Sorted Conv" := 4.0; END_IF;
   IF NOT "Base Exit Conveyor Green" THEN "Bases Green Sorted Conv" := 0.0; END_IF;
   IF "Base_Exit_conveyor_blue" THEN "Bases Blue Sorted Conv(1)" := -4.0; END_IF;
   IF NOT "Base_Exit_conveyor_blue" THEN "Bases Blue Sorted Conv(1)" := 0.0; END_IF;
   IF "Base_Exit_conveyor_blue" THEN "Bases Blue Sorted Conv(2)" := 4.0; END_IF;
   IF NOT "Base_Exit_conveyor_blue" THEN "Bases Blue Sorted Conv(2)" := 0.0; END_IF;
   IF "Base Exit Conveyor Green" THEN "Bases Green Sorted Conv(1)" := -4.0; END_IF;
   IF NOT "Base Exit Conveyor Green" THEN "Bases Green Sorted Conv(1)" := 0.0; END_IF;
   IF "Base Exit Conveyor Green" THEN "Bases Green Sorted Conv(2)" := 4.0; END_IF;
   IF NOT "Base Exit Conveyor Green" THEN "Bases Green Sorted Conv(2)" := 0.0; END_IF;
   IF "Base Exit Conveyor Green" THEN "Bases Green Sorted Conv(3)" := 4.0; END_IF;
   IF NOT "Base Exit Conveyor Green" THEN "Bases Green Sorted Conv(3)" := 0.0; END_IF;
   IF "Base Exit Conveyor Green" THEN "Bases Green Sorted Conv(4)" := 4.0; END_IF;
   IF NOT "Base Exit Conveyor Green" THEN "Bases Green Sorted Conv(4)" := 0.0; END_IF;
   IF "Base Exit Conveyor Green" THEN "Bases Green Sorted Conv(5)" := -4.0; END_IF;
   IF NOT "Base Exit Conveyor Green" THEN "Bases Green Sorted Conv(5)" := 0.0; END_IF;
   IF "Base Exit Conveyor Green" THEN "Bases Green Sorted Conv(6)" := 4.0; END_IF;
   IF NOT "Base Exit Conveyor Green" THEN "Bases Green Sorted Conv(6)" := 0.0; END_IF;
END_REGION

REGION Network 8
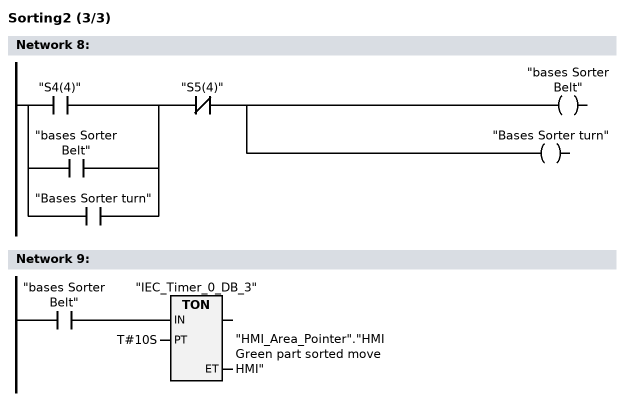
   RUNG wire#powerrail
      Contact( "S4(4)" )
      wire#w1
      I_Contact( "S5(4)" )
      wire#w2
      Coil( "bases Sorter  Belt" )
   END_RUNG
   RUNG wire#powerrail
      Contact( "bases Sorter  Belt" )
   END_RUNG wire#w1
   RUNG wire#powerrail
      Contact( "Bases Sorter turn" )
   END_RUNG wire#w1
   RUNG wire#w2
      Coil( "Bases Sorter turn" )
   END_RUNG
   // the same network as SCL:
   "bases Sorter  Belt" := ("S4(4)" OR "bases Sorter  Belt" OR "Bases Sorter turn") AND NOT "S5(4)";
   "Bases Sorter turn" := "bases Sorter  Belt";
END_REGION

REGION Network 9
   "IEC_Timer_0_DB_3".TON(IN := "bases Sorter  Belt",
                          PT := T#10S,
                          ET => "HMI_Area_Pointer"."HMI Green part sorted move HMI");
END_REGION
END_FUNCTION_BLOCK

FUNCTION_BLOCK "Assembler Blue"   // FB6, LAD
{ S7_Optimized_Access := 'TRUE' }
VERSION : 0.1
   VAR_TEMP   // added for the SCL form of the ladder/FBD networks
      _w1 : Bool;
      _w2 : Bool;
      _w3 : Bool;
      _w4 : Bool;
      _w5 : Bool;
      _w6 : Bool;
   END_VAR
BEGIN

REGION Network 1: States
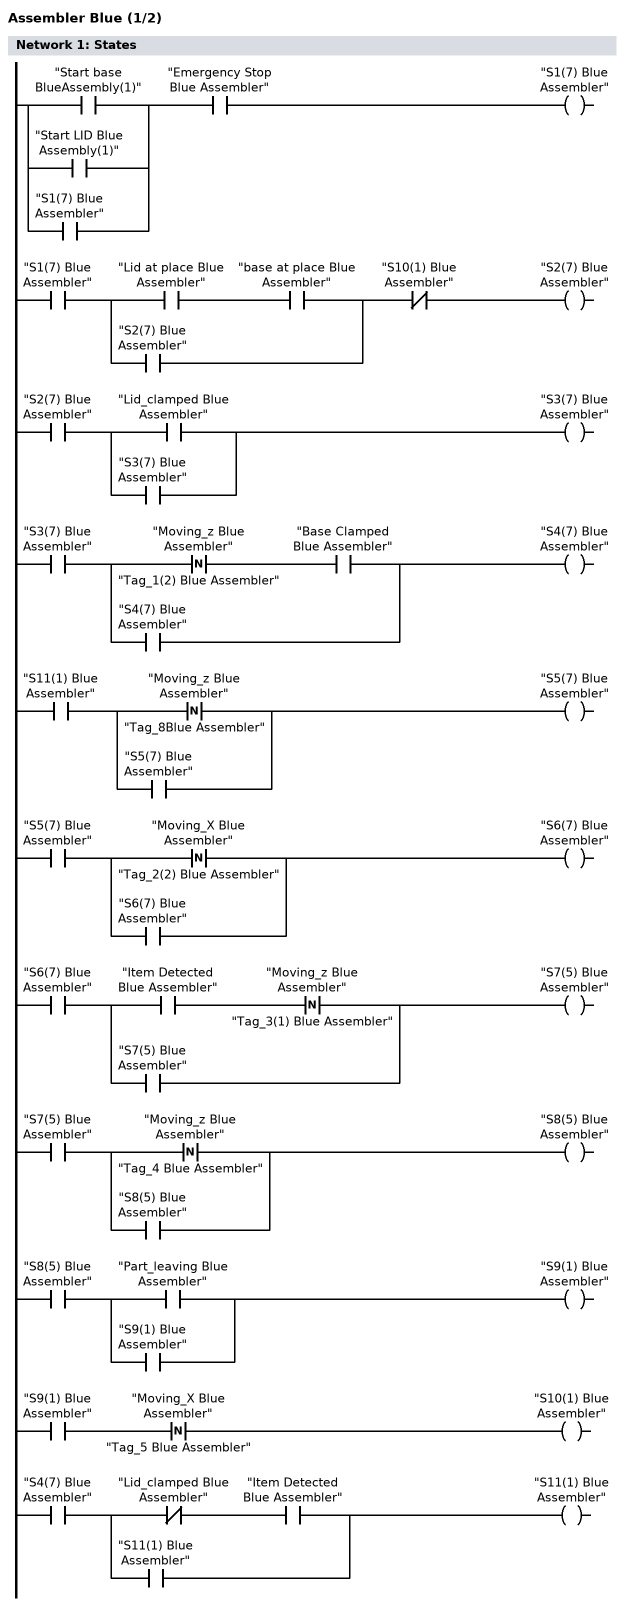
   RUNG wire#powerrail
      Contact( "Start base BlueAssembly(1)" )
      wire#w1
      Contact( "Emergency Stop Blue Assembler" )
      Coil( "S1(7) Blue Assembler" )
   END_RUNG
   RUNG wire#powerrail
      Contact( "Start LID Blue Assembly(1)" )
   END_RUNG wire#w1
   RUNG wire#powerrail
      Contact( "S1(7) Blue Assembler" )
   END_RUNG wire#w1
   RUNG wire#powerrail
      Contact( "S1(7) Blue Assembler" )
      wire#w2
      Contact( "Lid at place Blue Assembler" )
      Contact( "base at place Blue Assembler" )
      wire#w3
      I_Contact( "S10(1) Blue Assembler" )
      Coil( "S2(7) Blue Assembler" )
   END_RUNG
   RUNG wire#w2
      Contact( "S2(7) Blue Assembler" )
   END_RUNG wire#w3
   RUNG wire#powerrail
      Contact( "S2(7) Blue Assembler" )
      wire#w4
      Contact( "Lid_clamped Blue Assembler" )
      wire#w5
      Coil( "S3(7) Blue Assembler" )
   END_RUNG
   RUNG wire#w4
      Contact( "S3(7) Blue Assembler" )
   END_RUNG wire#w5
   RUNG wire#powerrail
      Contact( "S3(7) Blue Assembler" )
      wire#w6
      N_Contact(operand := "Moving_z Blue Assembler", bit := "Tag_1(2) Blue Assembler")
      Contact( "Base Clamped Blue Assembler" )
      wire#w7
      Coil( "S4(7) Blue Assembler" )
   END_RUNG
   RUNG wire#w6
      Contact( "S4(7) Blue Assembler" )
   END_RUNG wire#w7
   RUNG wire#powerrail
      Contact( "S11(1) Blue Assembler" )
      wire#w8
      N_Contact(operand := "Moving_z Blue Assembler", bit := "Tag_8Blue Assembler")
      wire#w9
      Coil( "S5(7) Blue Assembler" )
   END_RUNG
   RUNG wire#w8
      Contact( "S5(7) Blue Assembler" )
   END_RUNG wire#w9
   RUNG wire#powerrail
      Contact( "S5(7) Blue Assembler" )
      wire#w10
      N_Contact(operand := "Moving_X Blue Assembler", bit := "Tag_2(2) Blue Assembler")
      wire#w11
      Coil( "S6(7) Blue Assembler" )
   END_RUNG
   RUNG wire#w10
      Contact( "S6(7) Blue Assembler" )
   END_RUNG wire#w11
   RUNG wire#powerrail
      Contact( "S6(7) Blue Assembler" )
      wire#w12
      Contact( "Item Detected Blue Assembler" )
      N_Contact(operand := "Moving_z Blue Assembler", bit := "Tag_3(1) Blue Assembler")
      wire#w13
      Coil( "S7(5) Blue Assembler" )
   END_RUNG
   RUNG wire#w12
      Contact( "S7(5) Blue Assembler" )
   END_RUNG wire#w13
   RUNG wire#powerrail
      Contact( "S7(5) Blue Assembler" )
      wire#w14
      N_Contact(operand := "Moving_z Blue Assembler", bit := "Tag_4 Blue Assembler")
      wire#w15
      Coil( "S8(5) Blue Assembler" )
   END_RUNG
   RUNG wire#w14
      Contact( "S8(5) Blue Assembler" )
   END_RUNG wire#w15
   RUNG wire#powerrail
      Contact( "S8(5) Blue Assembler" )
      wire#w16
      Contact( "Part_leaving Blue Assembler" )
      wire#w17
      Coil( "S9(1) Blue Assembler" )
   END_RUNG
   RUNG wire#w16
      Contact( "S9(1) Blue Assembler" )
   END_RUNG wire#w17
   RUNG wire#powerrail
      Contact( "S9(1) Blue Assembler" )
      N_Contact(operand := "Moving_X Blue Assembler", bit := "Tag_5 Blue Assembler")
      Coil( "S10(1) Blue Assembler" )
   END_RUNG
   RUNG wire#powerrail
      Contact( "S4(7) Blue Assembler" )
      wire#w18
      I_Contact( "Lid_clamped Blue Assembler" )
      Contact( "Item Detected Blue Assembler" )
      wire#w19
      Coil( "S11(1) Blue Assembler" )
   END_RUNG
   RUNG wire#w18
      Contact( "S11(1) Blue Assembler" )
   END_RUNG wire#w19
   // the same network as SCL:
   "S1(7) Blue Assembler" := ("Start base BlueAssembly(1)" OR "Start LID Blue Assembly(1)" OR "S1(7) Blue Assembler") AND "Emergency Stop Blue Assembler";
   "S2(7) Blue Assembler" := "S1(7) Blue Assembler" AND (("Lid at place Blue Assembler" AND "base at place Blue Assembler") OR "S2(7) Blue Assembler") AND NOT "S10(1) Blue Assembler";
   "S3(7) Blue Assembler" := "S2(7) Blue Assembler" AND ("Lid_clamped Blue Assembler" OR "S3(7) Blue Assembler");
   #_w1 := "S3(7) Blue Assembler" AND NOT "Moving_z Blue Assembler" AND "Tag_1(2) Blue Assembler";   // falling edge of "Moving_z Blue Assembler"
   "Tag_1(2) Blue Assembler" := "Moving_z Blue Assembler";
   "S4(7) Blue Assembler" := (#_w1 AND "Base Clamped Blue Assembler") OR ("S3(7) Blue Assembler" AND "S4(7) Blue Assembler");
   #_w2 := "S11(1) Blue Assembler" AND NOT "Moving_z Blue Assembler" AND "Tag_8Blue Assembler";   // falling edge of "Moving_z Blue Assembler"
   "Tag_8Blue Assembler" := "Moving_z Blue Assembler";
   "S5(7) Blue Assembler" := #_w2 OR ("S11(1) Blue Assembler" AND "S5(7) Blue Assembler");
   #_w3 := "S5(7) Blue Assembler" AND NOT "Moving_X Blue Assembler" AND "Tag_2(2) Blue Assembler";   // falling edge of "Moving_X Blue Assembler"
   "Tag_2(2) Blue Assembler" := "Moving_X Blue Assembler";
   "S6(7) Blue Assembler" := #_w3 OR ("S5(7) Blue Assembler" AND "S6(7) Blue Assembler");
   #_w4 := "S6(7) Blue Assembler" AND "Item Detected Blue Assembler" AND NOT "Moving_z Blue Assembler" AND "Tag_3(1) Blue Assembler";   // falling edge of "Moving_z Blue Assembler"
   "Tag_3(1) Blue Assembler" := "Moving_z Blue Assembler";
   "S7(5) Blue Assembler" := #_w4 OR ("S6(7) Blue Assembler" AND "S7(5) Blue Assembler");
   #_w5 := "S7(5) Blue Assembler" AND NOT "Moving_z Blue Assembler" AND "Tag_4 Blue Assembler";   // falling edge of "Moving_z Blue Assembler"
   "Tag_4 Blue Assembler" := "Moving_z Blue Assembler";
   "S8(5) Blue Assembler" := #_w5 OR ("S7(5) Blue Assembler" AND "S8(5) Blue Assembler");
   "S9(1) Blue Assembler" := "S8(5) Blue Assembler" AND ("Part_leaving Blue Assembler" OR "S9(1) Blue Assembler");
   #_w6 := "S9(1) Blue Assembler" AND NOT "Moving_X Blue Assembler" AND "Tag_5 Blue Assembler";   // falling edge of "Moving_X Blue Assembler"
   "Tag_5 Blue Assembler" := "Moving_X Blue Assembler";
   "S10(1) Blue Assembler" := #_w6;
   "S11(1) Blue Assembler" := "S4(7) Blue Assembler" AND ((NOT "Lid_clamped Blue Assembler" AND "Item Detected Blue Assembler") OR "S11(1) Blue Assembler");
END_REGION

REGION Network 2: Actuators
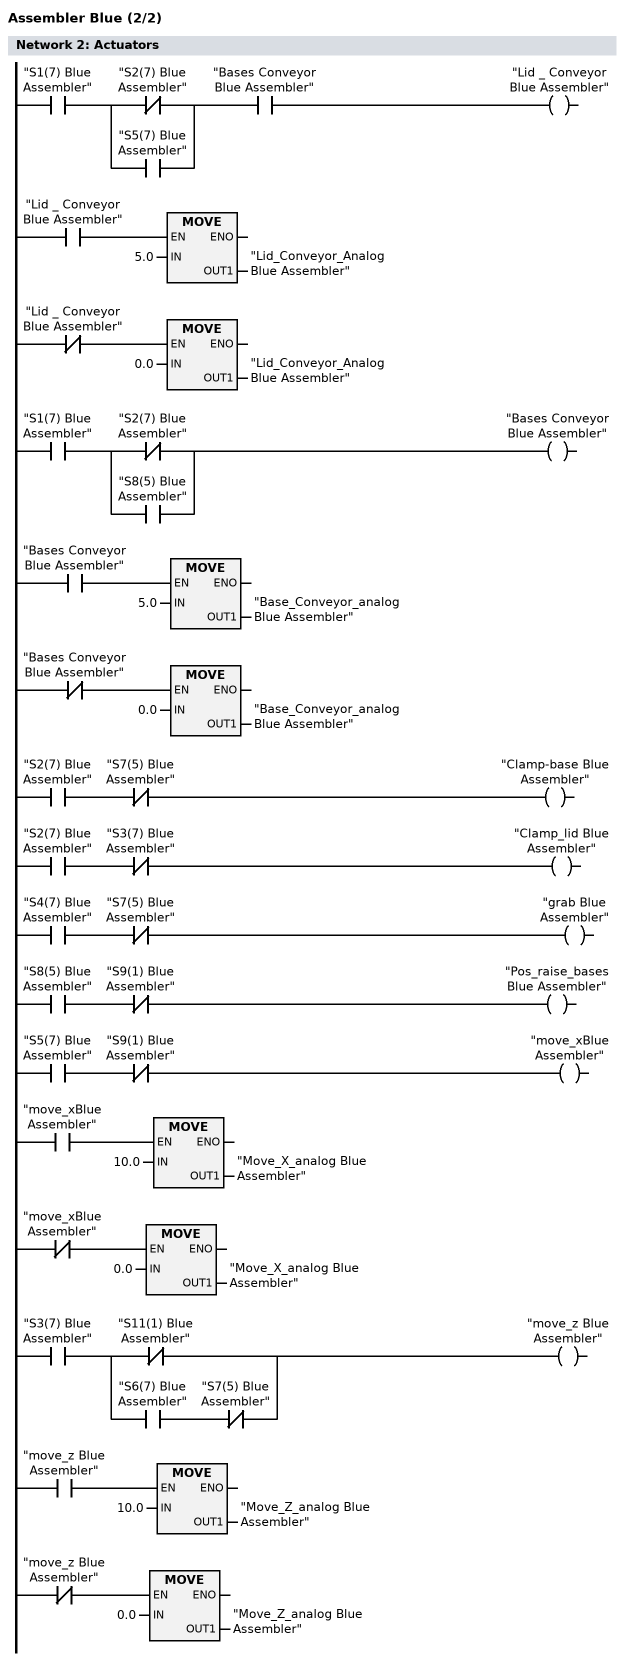
   RUNG wire#powerrail
      Contact( "S1(7) Blue Assembler" )
      wire#w1
      I_Contact( "S2(7) Blue Assembler" )
      wire#w2
      Contact( "Bases Conveyor Blue Assembler" )
      Coil( "Lid _ Conveyor Blue Assembler" )
   END_RUNG
   RUNG wire#w1
      Contact( "S5(7) Blue Assembler" )
   END_RUNG wire#w2
   RUNG wire#powerrail
      Contact( "Lid _ Conveyor Blue Assembler" )
      Move(in := 5.0, out1 => "Lid_Conveyor_Analog Blue Assembler")
   END_RUNG
   RUNG wire#powerrail
      I_Contact( "Lid _ Conveyor Blue Assembler" )
      Move(in := 0.0, out1 => "Lid_Conveyor_Analog Blue Assembler")
   END_RUNG
   RUNG wire#powerrail
      Contact( "S1(7) Blue Assembler" )
      wire#w3
      I_Contact( "S2(7) Blue Assembler" )
      wire#w4
      Coil( "Bases Conveyor Blue Assembler" )
   END_RUNG
   RUNG wire#w3
      Contact( "S8(5) Blue Assembler" )
   END_RUNG wire#w4
   RUNG wire#powerrail
      Contact( "Bases Conveyor Blue Assembler" )
      Move(in := 5.0, out1 => "Base_Conveyor_analog Blue Assembler")
   END_RUNG
   RUNG wire#powerrail
      I_Contact( "Bases Conveyor Blue Assembler" )
      Move(in := 0.0, out1 => "Base_Conveyor_analog Blue Assembler")
   END_RUNG
   RUNG wire#powerrail
      Contact( "S2(7) Blue Assembler" )
      I_Contact( "S7(5) Blue Assembler" )
      Coil( "Clamp-base Blue Assembler" )
   END_RUNG
   RUNG wire#powerrail
      Contact( "S2(7) Blue Assembler" )
      I_Contact( "S3(7) Blue Assembler" )
      Coil( "Clamp_lid Blue Assembler" )
   END_RUNG
   RUNG wire#powerrail
      Contact( "S4(7) Blue Assembler" )
      I_Contact( "S7(5) Blue Assembler" )
      Coil( "grab Blue Assembler" )
   END_RUNG
   RUNG wire#powerrail
      Contact( "S8(5) Blue Assembler" )
      I_Contact( "S9(1) Blue Assembler" )
      Coil( "Pos_raise_bases Blue Assembler" )
   END_RUNG
   RUNG wire#powerrail
      Contact( "S5(7) Blue Assembler" )
      I_Contact( "S9(1) Blue Assembler" )
      Coil( "move_xBlue Assembler" )
   END_RUNG
   RUNG wire#powerrail
      Contact( "move_xBlue Assembler" )
      Move(in := 10.0, out1 => "Move_X_analog Blue Assembler")
   END_RUNG
   RUNG wire#powerrail
      I_Contact( "move_xBlue Assembler" )
      Move(in := 0.0, out1 => "Move_X_analog Blue Assembler")
   END_RUNG
   RUNG wire#powerrail
      Contact( "S3(7) Blue Assembler" )
      wire#w5
      I_Contact( "S11(1) Blue Assembler" )
      wire#w6
      Coil( "move_z Blue Assembler" )
   END_RUNG
   RUNG wire#w5
      Contact( "S6(7) Blue Assembler" )
      I_Contact( "S7(5) Blue Assembler" )
   END_RUNG wire#w6
   RUNG wire#powerrail
      Contact( "move_z Blue Assembler" )
      Move(in := 10.0, out1 => "Move_Z_analog Blue Assembler")
   END_RUNG
   RUNG wire#powerrail
      I_Contact( "move_z Blue Assembler" )
      Move(in := 0.0, out1 => "Move_Z_analog Blue Assembler")
   END_RUNG
   // the same network as SCL:
   "Lid _ Conveyor Blue Assembler" := "S1(7) Blue Assembler" AND (NOT "S2(7) Blue Assembler" OR "S5(7) Blue Assembler") AND "Bases Conveyor Blue Assembler";
   IF "Lid _ Conveyor Blue Assembler" THEN "Lid_Conveyor_Analog Blue Assembler" := 5.0; END_IF;
   IF NOT "Lid _ Conveyor Blue Assembler" THEN "Lid_Conveyor_Analog Blue Assembler" := 0.0; END_IF;
   "Bases Conveyor Blue Assembler" := "S1(7) Blue Assembler" AND (NOT "S2(7) Blue Assembler" OR "S8(5) Blue Assembler");
   IF "Bases Conveyor Blue Assembler" THEN "Base_Conveyor_analog Blue Assembler" := 5.0; END_IF;
   IF NOT "Bases Conveyor Blue Assembler" THEN "Base_Conveyor_analog Blue Assembler" := 0.0; END_IF;
   "Clamp-base Blue Assembler" := "S2(7) Blue Assembler" AND NOT "S7(5) Blue Assembler";
   "Clamp_lid Blue Assembler" := "S2(7) Blue Assembler" AND NOT "S3(7) Blue Assembler";
   "grab Blue Assembler" := "S4(7) Blue Assembler" AND NOT "S7(5) Blue Assembler";
   "Pos_raise_bases Blue Assembler" := "S8(5) Blue Assembler" AND NOT "S9(1) Blue Assembler";
   "move_xBlue Assembler" := "S5(7) Blue Assembler" AND NOT "S9(1) Blue Assembler";
   IF "move_xBlue Assembler" THEN "Move_X_analog Blue Assembler" := 10.0; END_IF;
   IF NOT "move_xBlue Assembler" THEN "Move_X_analog Blue Assembler" := 0.0; END_IF;
   "move_z Blue Assembler" := "S3(7) Blue Assembler" AND (NOT "S11(1) Blue Assembler" OR ("S6(7) Blue Assembler" AND NOT "S7(5) Blue Assembler"));
   IF "move_z Blue Assembler" THEN "Move_Z_analog Blue Assembler" := 10.0; END_IF;
   IF NOT "move_z Blue Assembler" THEN "Move_Z_analog Blue Assembler" := 0.0; END_IF;
END_REGION
END_FUNCTION_BLOCK

FUNCTION_BLOCK "Assembler Green"   // FB7, LAD
{ S7_Optimized_Access := 'TRUE' }
VERSION : 0.1
   VAR_TEMP   // added for the SCL form of the ladder/FBD networks
      _w1 : Bool;
      _w2 : Bool;
      _w3 : Bool;
      _w4 : Bool;
      _w5 : Bool;
      _w6 : Bool;
   END_VAR
BEGIN

REGION Network 1: States
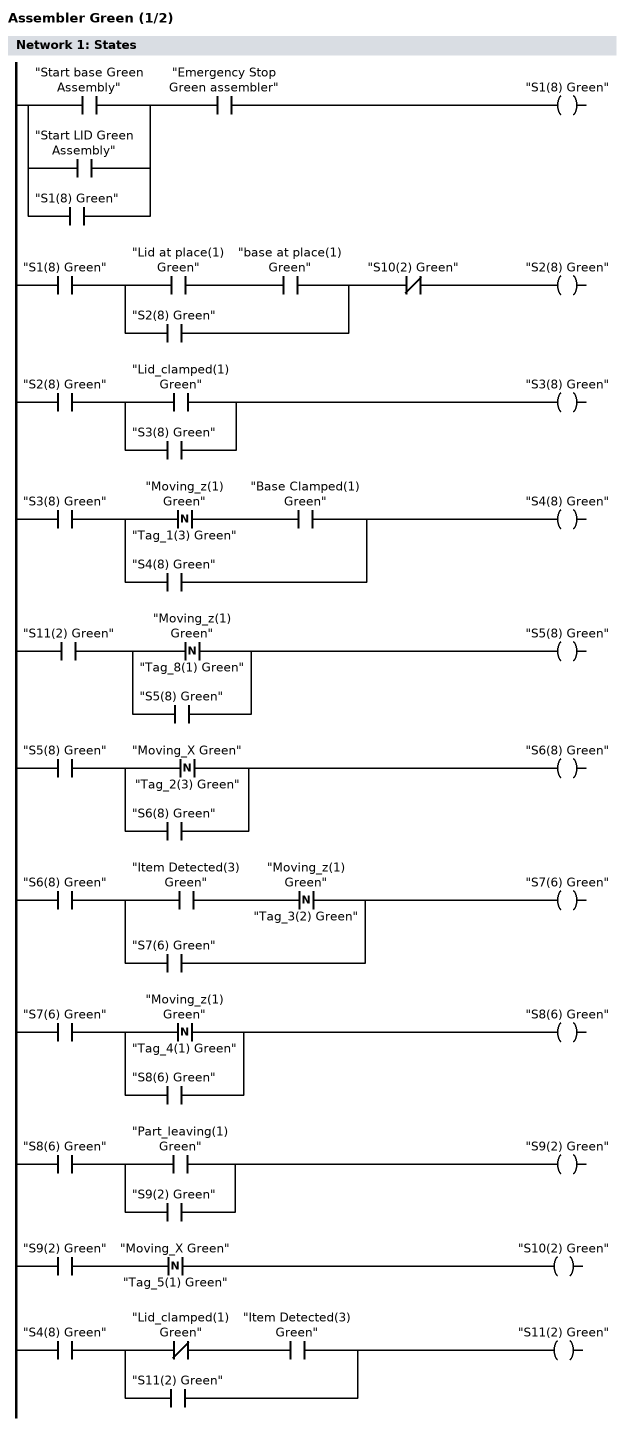
   RUNG wire#powerrail
      Contact( "Start base Green Assembly" )
      wire#w1
      Contact( "Emergency Stop Green assembler" )
      Coil( "S1(8) Green" )
   END_RUNG
   RUNG wire#powerrail
      Contact( "Start LID Green Assembly" )
   END_RUNG wire#w1
   RUNG wire#powerrail
      Contact( "S1(8) Green" )
   END_RUNG wire#w1
   RUNG wire#powerrail
      Contact( "S1(8) Green" )
      wire#w2
      Contact( "Lid at place(1) Green" )
      Contact( "base at place(1) Green" )
      wire#w3
      I_Contact( "S10(2) Green" )
      Coil( "S2(8) Green" )
   END_RUNG
   RUNG wire#w2
      Contact( "S2(8) Green" )
   END_RUNG wire#w3
   RUNG wire#powerrail
      Contact( "S2(8) Green" )
      wire#w4
      Contact( "Lid_clamped(1) Green" )
      wire#w5
      Coil( "S3(8) Green" )
   END_RUNG
   RUNG wire#w4
      Contact( "S3(8) Green" )
   END_RUNG wire#w5
   RUNG wire#powerrail
      Contact( "S3(8) Green" )
      wire#w6
      N_Contact(operand := "Moving_z(1) Green", bit := "Tag_1(3) Green")
      Contact( "Base Clamped(1) Green" )
      wire#w7
      Coil( "S4(8) Green" )
   END_RUNG
   RUNG wire#w6
      Contact( "S4(8) Green" )
   END_RUNG wire#w7
   RUNG wire#powerrail
      Contact( "S11(2) Green" )
      wire#w8
      N_Contact(operand := "Moving_z(1) Green", bit := "Tag_8(1) Green")
      wire#w9
      Coil( "S5(8) Green" )
   END_RUNG
   RUNG wire#w8
      Contact( "S5(8) Green" )
   END_RUNG wire#w9
   RUNG wire#powerrail
      Contact( "S5(8) Green" )
      wire#w10
      N_Contact(operand := "Moving_X Green", bit := "Tag_2(3) Green")
      wire#w11
      Coil( "S6(8) Green" )
   END_RUNG
   RUNG wire#w10
      Contact( "S6(8) Green" )
   END_RUNG wire#w11
   RUNG wire#powerrail
      Contact( "S6(8) Green" )
      wire#w12
      Contact( "Item Detected(3) Green" )
      N_Contact(operand := "Moving_z(1) Green", bit := "Tag_3(2) Green")
      wire#w13
      Coil( "S7(6) Green" )
   END_RUNG
   RUNG wire#w12
      Contact( "S7(6) Green" )
   END_RUNG wire#w13
   RUNG wire#powerrail
      Contact( "S7(6) Green" )
      wire#w14
      N_Contact(operand := "Moving_z(1) Green", bit := "Tag_4(1) Green")
      wire#w15
      Coil( "S8(6) Green" )
   END_RUNG
   RUNG wire#w14
      Contact( "S8(6) Green" )
   END_RUNG wire#w15
   RUNG wire#powerrail
      Contact( "S8(6) Green" )
      wire#w16
      Contact( "Part_leaving(1) Green" )
      wire#w17
      Coil( "S9(2) Green" )
   END_RUNG
   RUNG wire#w16
      Contact( "S9(2) Green" )
   END_RUNG wire#w17
   RUNG wire#powerrail
      Contact( "S9(2) Green" )
      N_Contact(operand := "Moving_X Green", bit := "Tag_5(1) Green")
      Coil( "S10(2) Green" )
   END_RUNG
   RUNG wire#powerrail
      Contact( "S4(8) Green" )
      wire#w18
      I_Contact( "Lid_clamped(1) Green" )
      Contact( "Item Detected(3) Green" )
      wire#w19
      Coil( "S11(2) Green" )
   END_RUNG
   RUNG wire#w18
      Contact( "S11(2) Green" )
   END_RUNG wire#w19
   // the same network as SCL:
   "S1(8) Green" := ("Start base Green Assembly" OR "Start LID Green Assembly" OR "S1(8) Green") AND "Emergency Stop Green assembler";
   "S2(8) Green" := "S1(8) Green" AND (("Lid at place(1) Green" AND "base at place(1) Green") OR "S2(8) Green") AND NOT "S10(2) Green";
   "S3(8) Green" := "S2(8) Green" AND ("Lid_clamped(1) Green" OR "S3(8) Green");
   #_w1 := "S3(8) Green" AND NOT "Moving_z(1) Green" AND "Tag_1(3) Green";   // falling edge of "Moving_z(1) Green"
   "Tag_1(3) Green" := "Moving_z(1) Green";
   "S4(8) Green" := (#_w1 AND "Base Clamped(1) Green") OR ("S3(8) Green" AND "S4(8) Green");
   #_w2 := "S11(2) Green" AND NOT "Moving_z(1) Green" AND "Tag_8(1) Green";   // falling edge of "Moving_z(1) Green"
   "Tag_8(1) Green" := "Moving_z(1) Green";
   "S5(8) Green" := #_w2 OR ("S11(2) Green" AND "S5(8) Green");
   #_w3 := "S5(8) Green" AND NOT "Moving_X Green" AND "Tag_2(3) Green";   // falling edge of "Moving_X Green"
   "Tag_2(3) Green" := "Moving_X Green";
   "S6(8) Green" := #_w3 OR ("S5(8) Green" AND "S6(8) Green");
   #_w4 := "S6(8) Green" AND "Item Detected(3) Green" AND NOT "Moving_z(1) Green" AND "Tag_3(2) Green";   // falling edge of "Moving_z(1) Green"
   "Tag_3(2) Green" := "Moving_z(1) Green";
   "S7(6) Green" := #_w4 OR ("S6(8) Green" AND "S7(6) Green");
   #_w5 := "S7(6) Green" AND NOT "Moving_z(1) Green" AND "Tag_4(1) Green";   // falling edge of "Moving_z(1) Green"
   "Tag_4(1) Green" := "Moving_z(1) Green";
   "S8(6) Green" := #_w5 OR ("S7(6) Green" AND "S8(6) Green");
   "S9(2) Green" := "S8(6) Green" AND ("Part_leaving(1) Green" OR "S9(2) Green");
   #_w6 := "S9(2) Green" AND NOT "Moving_X Green" AND "Tag_5(1) Green";   // falling edge of "Moving_X Green"
   "Tag_5(1) Green" := "Moving_X Green";
   "S10(2) Green" := #_w6;
   "S11(2) Green" := "S4(8) Green" AND ((NOT "Lid_clamped(1) Green" AND "Item Detected(3) Green") OR "S11(2) Green");
END_REGION

REGION Network 2: Actuators
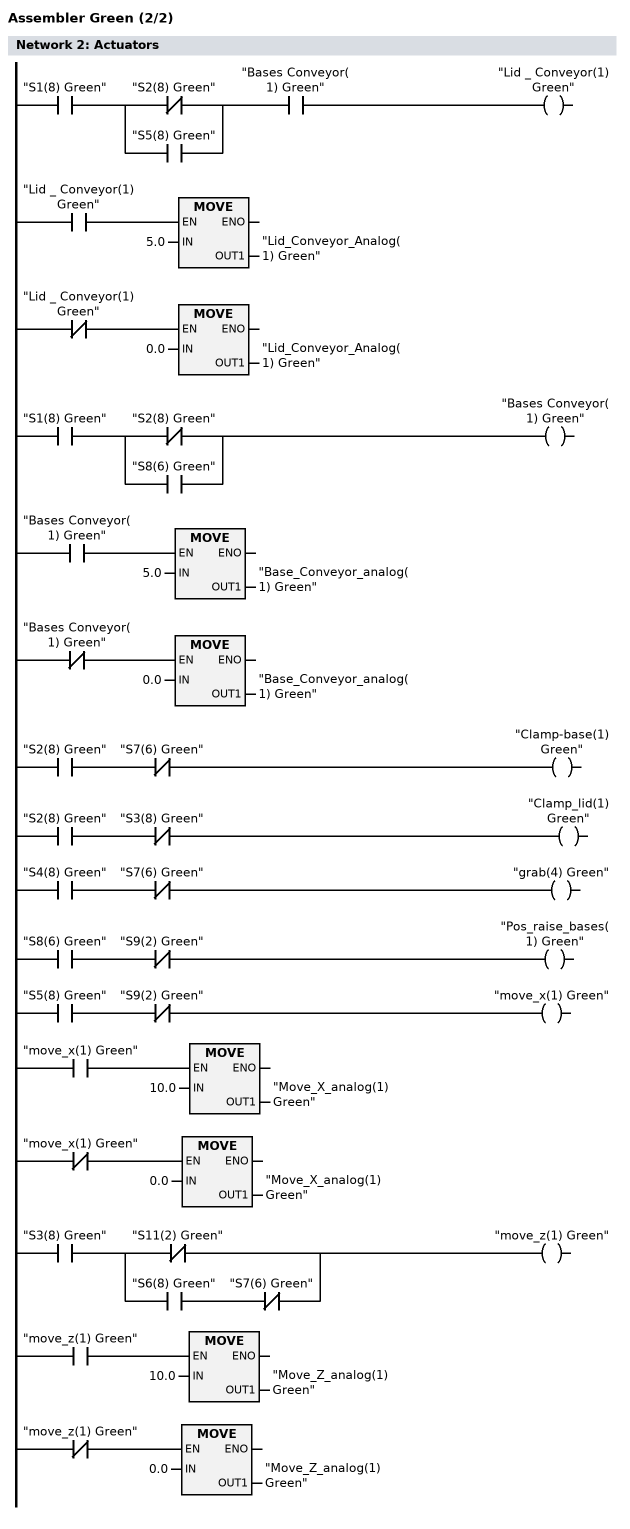
   RUNG wire#powerrail
      Contact( "S1(8) Green" )
      wire#w1
      I_Contact( "S2(8) Green" )
      wire#w2
      Contact( "Bases Conveyor(1) Green" )
      Coil( "Lid _ Conveyor(1) Green" )
   END_RUNG
   RUNG wire#w1
      Contact( "S5(8) Green" )
   END_RUNG wire#w2
   RUNG wire#powerrail
      Contact( "Lid _ Conveyor(1) Green" )
      Move(in := 5.0, out1 => "Lid_Conveyor_Analog(1) Green")
   END_RUNG
   RUNG wire#powerrail
      I_Contact( "Lid _ Conveyor(1) Green" )
      Move(in := 0.0, out1 => "Lid_Conveyor_Analog(1) Green")
   END_RUNG
   RUNG wire#powerrail
      Contact( "S1(8) Green" )
      wire#w3
      I_Contact( "S2(8) Green" )
      wire#w4
      Coil( "Bases Conveyor(1) Green" )
   END_RUNG
   RUNG wire#w3
      Contact( "S8(6) Green" )
   END_RUNG wire#w4
   RUNG wire#powerrail
      Contact( "Bases Conveyor(1) Green" )
      Move(in := 5.0, out1 => "Base_Conveyor_analog(1) Green")
   END_RUNG
   RUNG wire#powerrail
      I_Contact( "Bases Conveyor(1) Green" )
      Move(in := 0.0, out1 => "Base_Conveyor_analog(1) Green")
   END_RUNG
   RUNG wire#powerrail
      Contact( "S2(8) Green" )
      I_Contact( "S7(6) Green" )
      Coil( "Clamp-base(1) Green" )
   END_RUNG
   RUNG wire#powerrail
      Contact( "S2(8) Green" )
      I_Contact( "S3(8) Green" )
      Coil( "Clamp_lid(1) Green" )
   END_RUNG
   RUNG wire#powerrail
      Contact( "S4(8) Green" )
      I_Contact( "S7(6) Green" )
      Coil( "grab(4) Green" )
   END_RUNG
   RUNG wire#powerrail
      Contact( "S8(6) Green" )
      I_Contact( "S9(2) Green" )
      Coil( "Pos_raise_bases(1) Green" )
   END_RUNG
   RUNG wire#powerrail
      Contact( "S5(8) Green" )
      I_Contact( "S9(2) Green" )
      Coil( "move_x(1) Green" )
   END_RUNG
   RUNG wire#powerrail
      Contact( "move_x(1) Green" )
      Move(in := 10.0, out1 => "Move_X_analog(1) Green")
   END_RUNG
   RUNG wire#powerrail
      I_Contact( "move_x(1) Green" )
      Move(in := 0.0, out1 => "Move_X_analog(1) Green")
   END_RUNG
   RUNG wire#powerrail
      Contact( "S3(8) Green" )
      wire#w5
      I_Contact( "S11(2) Green" )
      wire#w6
      Coil( "move_z(1) Green" )
   END_RUNG
   RUNG wire#w5
      Contact( "S6(8) Green" )
      I_Contact( "S7(6) Green" )
   END_RUNG wire#w6
   RUNG wire#powerrail
      Contact( "move_z(1) Green" )
      Move(in := 10.0, out1 => "Move_Z_analog(1) Green")
   END_RUNG
   RUNG wire#powerrail
      I_Contact( "move_z(1) Green" )
      Move(in := 0.0, out1 => "Move_Z_analog(1) Green")
   END_RUNG
   // the same network as SCL:
   "Lid _ Conveyor(1) Green" := "S1(8) Green" AND (NOT "S2(8) Green" OR "S5(8) Green") AND "Bases Conveyor(1) Green";
   IF "Lid _ Conveyor(1) Green" THEN "Lid_Conveyor_Analog(1) Green" := 5.0; END_IF;
   IF NOT "Lid _ Conveyor(1) Green" THEN "Lid_Conveyor_Analog(1) Green" := 0.0; END_IF;
   "Bases Conveyor(1) Green" := "S1(8) Green" AND (NOT "S2(8) Green" OR "S8(6) Green");
   IF "Bases Conveyor(1) Green" THEN "Base_Conveyor_analog(1) Green" := 5.0; END_IF;
   IF NOT "Bases Conveyor(1) Green" THEN "Base_Conveyor_analog(1) Green" := 0.0; END_IF;
   "Clamp-base(1) Green" := "S2(8) Green" AND NOT "S7(6) Green";
   "Clamp_lid(1) Green" := "S2(8) Green" AND NOT "S3(8) Green";
   "grab(4) Green" := "S4(8) Green" AND NOT "S7(6) Green";
   "Pos_raise_bases(1) Green" := "S8(6) Green" AND NOT "S9(2) Green";
   "move_x(1) Green" := "S5(8) Green" AND NOT "S9(2) Green";
   IF "move_x(1) Green" THEN "Move_X_analog(1) Green" := 10.0; END_IF;
   IF NOT "move_x(1) Green" THEN "Move_X_analog(1) Green" := 0.0; END_IF;
   "move_z(1) Green" := "S3(8) Green" AND (NOT "S11(2) Green" OR ("S6(8) Green" AND NOT "S7(6) Green"));
   IF "move_z(1) Green" THEN "Move_Z_analog(1) Green" := 10.0; END_IF;
   IF NOT "move_z(1) Green" THEN "Move_Z_analog(1) Green" := 0.0; END_IF;
END_REGION
END_FUNCTION_BLOCK

ORGANIZATION_BLOCK "Main"   // OB1, LAD, ProgramCycle
TITLE = "Main Program Sweep (Cycle)"
{ S7_Optimized_Access := 'TRUE' }
VERSION : 0.1
   VAR_INPUT
      Initial_Call : Bool;   // Initial call of this OB
      Remanence : Bool;   // =True, if remanent data are available
   END_VAR
BEGIN

REGION Network 1
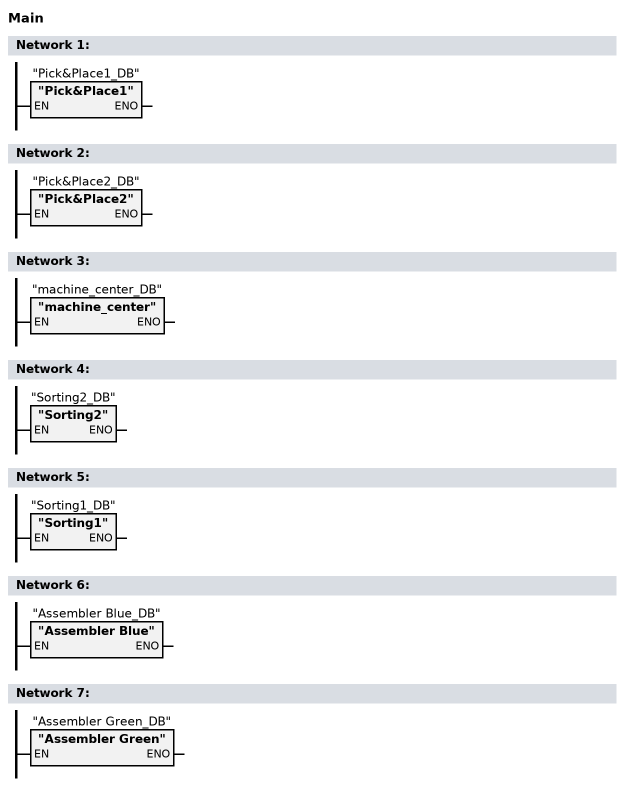
   RUNG wire#powerrail
      "Pick&Place1_DB"()
   END_RUNG
   // the same network as SCL:
   "Pick&Place1_DB"();   // "Pick&Place1"
END_REGION

REGION Network 2
   RUNG wire#powerrail
      "Pick&Place2_DB"()
   END_RUNG
   // the same network as SCL:
   "Pick&Place2_DB"();   // "Pick&Place2"
END_REGION

REGION Network 3
   RUNG wire#powerrail
      "machine_center_DB"()
   END_RUNG
   // the same network as SCL:
   "machine_center_DB"();   // "machine_center"
END_REGION

REGION Network 4
   RUNG wire#powerrail
      "Sorting2_DB"()
   END_RUNG
   // the same network as SCL:
   "Sorting2_DB"();   // "Sorting2"
END_REGION

REGION Network 5
   RUNG wire#powerrail
      "Sorting1_DB"()
   END_RUNG
   // the same network as SCL:
   "Sorting1_DB"();   // "Sorting1"
END_REGION

REGION Network 6
   RUNG wire#powerrail
      "Assembler Blue_DB"()
   END_RUNG
   // the same network as SCL:
   "Assembler Blue_DB"();   // "Assembler Blue"
END_REGION

REGION Network 7
   RUNG wire#powerrail
      "Assembler Green_DB"()
   END_RUNG
   // the same network as SCL:
   "Assembler Green_DB"();   // "Assembler Green"
END_REGION
END_ORGANIZATION_BLOCK

(* ===== HMI "HMI_RT_1" =====
system functions are stored by id; their names below are inferred from use
connection "HMI_Connection_1": ETHERNET, S7_1500_OMS

HMI tags "Default tag table"
   "Tag_ScreenNumber" : UInt, internal
   "HMI Assembly input part 1 Move" : Int, internal
   "HMI Assembly input part 2 Move" : Int, internal
   "HMI Assembly output part move" : Int, internal
   "HMI Blue part sorted move HMI" : DWord = PLC HMI_Area_Pointer."HMI blue part sorted move HMI" AT %DB1.DBW0, 1 s
   "HMI Broken_Sensor" : Int, internal
   "HMI Emergency stop system" : Bool = PLC Reset AT %I0.4, 1 s
   "HMI Entry_conveyor" : Bool = PLC Entry_conveyor AT %Q5.0, 1 s
   "HMI Grab" : Bool = PLC Grab AT %Q0.4, 1 s
   "HMI Green part sorted move HMI" : DWord = PLC HMI_Area_Pointer."HMI Green part sorted move HMI" AT %DB1.DBW0, 1 s
   "HMI Start system" : Bool = PLC "Start Button" AT %I0.3, 1 s
   "HMI Stop system" : Bool = PLC Stop AT %I0.5, 1 s
   "HMI_AREA_POINTER_Start PB" : Bool = PLC HMI_Area_Pointer."Start Whole System PB", 1 s
   "HMI_AREA_POINTER_Stop PB" : Bool = PLC HMI_Area_Pointer."Stop Whole System PB", 1 s
   "HMI_Box_Pick_and_place1" : DWord = PLC HMI_Area_Pointer.HMI_Box_Pick_and_place1, 1 s
   "HMI_Box_Pick_and_place2" : DWord = PLC HMI_Area_Pointer.HMI_Box_Pick_and_place2, 1 s
   "Machine center part before machining move" : Int, internal
   "Machining Center part after maching move" : Int, internal
   "s1" : Bool = PLC s1 AT %M92.0, 1 s
   "LID sorter Belt" : Bool = PLC "LID sorter Belt" AT %Q1.4, 1 s
   "LID green Sorted Conv ANalog" : Real = PLC "LID green Sorted Conv ANalog" AT %QD94, 1 s
   "LID sorting conveyor 1" : Real = PLC "LID sorting conveyor 1" AT %QD78, 1 s
   "Entry Conveyor 1" : Real = PLC "Entry Conveyor 1" AT %QD30, 1 s
   "Exit_Conveyor 1" : Real = PLC "Exit_Conveyor 1" AT %QD34, 1 s
   "Exit conveyor" : Bool = PLC "Exit conveyor" AT %Q5.1, 1 s
   "Lids_center_busy" : Bool = PLC Lids_center_busy AT %I1.7, 1 s
   "bases_center_busy" : Bool = PLC bases_center_busy AT %I2.3, 1 s
   "Bases_raw_conveyor" : Bool = PLC Bases_raw_conveyor AT %M73.0, 1 s
   "Exit_Conveyor" : Bool = PLC Exit_Conveyor AT %Q11.6, 1 s
   "bases Sorter  Belt" : Bool = PLC "bases Sorter  Belt" AT %Q1.6, 1 s
   "S2(8) Green" : Bool = PLC "S2(8) Green" AT %M131.0, 1 s
   "S2(7) Blue Assembler" : Bool = PLC "S2(7) Blue Assembler" AT %M122.0, 1 s

discrete alarms
   1: 'please Repair', class Warnings, trigger "HMI Broken_Sensor" bit 0

Template "Template_1" 800x420
   Button "Exit" at 720,360 size 78x58; TextOff 'Exit'; PictureOff "ExitRuntime_TP700_Comfort_TR"; PictureOn "ExitRuntime_TP700_Comfort_TR"
      on Release: StopRuntime(0)
   Button "Template_Button" at 640,360 size 78x58; TextOff 'Text'
   Button "Template_Button_1" at 560,360 size 78x58; TextOff 'Text'
   Button "Template_Button_2" at 480,360 size 78x58; TextOff 'Text'
   Button "Template_Button_3" at 400,360 size 78x58; TextOff 'Text'
   Button "Template_Button_4" at 321,360 size 78x58; TextOff 'Text'
   Button "Template_Button_5" at 241,360 size 78x58; TextOff 'Text'
   Button "Template_Button_6" at 161,360 size 78x58; TextOff 'Text'
   Button "Alarms" at 81,360 size 78x58; TextOff 'Alarms'; PictureOff "AlarmDisplay_TP700_Comfort_TR"; PictureOn "AlarmDisplay_TP700_Comfort_TR"
      on Release: function_ef3f5d25("Alarm window_Unacknowledged", -1)
   Button "Start screen" at 1,360 size 78x58; TextOff 'Start screen'; PictureOff "NavigateHome_TP700_Comfort_TR"; PictureOn "NavigateHome_TP700_Comfort_TR"

screen "Alarm" 800x420
   AlarmView "Alarm view_1" at 63,36 size 689x300
   Button "Button_1" at 26,411 size 148x57; TextOff 'Broken Sensor'
      on Press: function_b14e0dd5("HMI Broken_Sensor", 0)
   Button "Button_2" at 442,352 size 122x34; TextOn 'Pick&Place'; TextOff 'Pick&Place'
      on Click: ActivateScreen("Pick&Place", 0)
   Button "Button_3" at 214,353 size 192x32; TextOn 'Sorting'; TextOff 'Sorting'
      on Click: ActivateScreen("Sorting", 0)
   Button "Button_4" at 201,425 size 192x32; TextOn 'Assembly'; TextOff 'Assembly'
      on Click: ActivateScreen("Assembly", 0)
   Button "Button_5" at 0,354 size 192x32; TextOn 'Main Screen'; TextOff 'Main Screen'
      on Click: ActivateScreen("Main Screen", 0)
   Button "Button_6" at 434,425 size 192x32; TextOn 'Machine Center'; TextOff 'Machine Center'
      on Click: ActivateScreen("Machine Center", 0)
   Button "Button_7" at 593,353 size 192x32; TextOn 'Sorting'; TextOff 'Sorting'
      on Click: ActivateScreen("Sorting", 0)

screen "Assembly" 800x420
   Button "Button_4" at 29,11 size 167x59; TextOn 'Stopped'; TextOff 'Emergency Stop'
      on Release: ResetBit("HMI_AREA_POINTER_Stop PB")
      on Press: SetBit("HMI_AREA_POINTER_Stop PB")
   GraphicView "Graphic view_1" at 443,260 size 330x46; Picture "Graphic_7"
   GraphicView "Graphic view_2" at 50,212 size 332x53; Picture "Graphic_7"
   Button "Button_1" at 344,70 size 99x33; TextOn 'Alarm'; TextOff 'Alarm'
      on Click: ActivateScreen("Alarm", 0)
   Button "Button_2" at 506,110 size 192x32; TextOn 'Sorting'; TextOff 'Sorting'
      on Click: ActivateScreen("Sorting", 0)
   GraphicView "Graphic view_4" at 48,329 size 332x53; Picture "Graphic_7"
   GraphicView "Graphic view_5" at 55,165 size 75x75; Picture "Graphic_13"
      HorizontalMovement <- "HMI Assembly input part 1 Move"
   GraphicView "Graphic view_6" at 80,269 size 75x75; Picture "Graphic_16"
      HorizontalMovement <- "HMI Assembly input part 2 Move"
   GraphicView "Graphic view_7" at 482,220 size 75x75; Picture "Graphic_17"
      HorizontalMovement <- "HMI Assembly output part move"
   Button "Button_7" at 260,19 size 242x35; TextOn 'Started'; TextOff 'Assembly Station'
      on Release: ResetBit("HMI_AREA_POINTER_Start PB")
      on Press: SetBit("HMI_AREA_POINTER_Start PB")
   Button "Button_5" at 506,70 size 192x32; TextOn 'Machine Center'; TextOff 'Machine Center'
      on Click: ActivateScreen("Machine Center", 0)
   Button "Button_6" at 300,110 size 192x32; TextOn 'Pick&Place'; TextOff 'Pick&Place'
      on Click: ActivateScreen("Pick&Place", 0)
   Button "Button_3" at 36,84 size 200x58; TextOn 'Main Screen'; TextOff 'Main Screen'
      on Click: ActivateScreen("Main Screen", 0)
   Circle "Circle_1" at 707,367 size 40x40
      Appearance <- "S2(8) Green"
   TextField "Text field_6" at 492,319 size 196x32; Text 'Assembly Blue'
   TextField "Text field_7" at 494,363 size 215x32; Text 'Assembly Green'
   Circle "Circle_2" at 707,323 size 40x40
      Appearance <- "S2(7) Blue Assembler"

screen "Machine Center" 800x420
   Button "Button_3" at 67,7 size 105x48; TextOn 'Started'; TextOff 'Start'
      on Release: ResetBit("HMI_AREA_POINTER_Start PB")
      on Press: SetBit("HMI_AREA_POINTER_Start PB")
   Button "Button_4" at 69,76 size 102x38; TextOn 'Stopped'; TextOff 'Stop'
      on Release: ResetBit("HMI_AREA_POINTER_Stop PB")
      on Press: SetBit("HMI_AREA_POINTER_Stop PB")
   GraphicView "Graphic view_1" at 431,265 size 330x46; Picture "Graphic_7"
   GraphicView "Graphic view_2" at 80,254 size 332x53; Picture "Graphic_7"
   Button "Button_1" at 321,113 size 99x33; TextOn 'Alarm'; TextOff 'Alarm'
      on Click: ActivateScreen("Alarm", 0)
   Button "Button_2" at 292,163 size 192x32; TextOn 'Sorting'; TextOff 'Sorting'
      on Click: ActivateScreen("Sorting", 0)
   GraphicView "Graphic view_4" at 117,219 size 75x75; Picture "Graphic_13"
      HorizontalMovement <- "Machine center part before machining move"
   GraphicView "Graphic view_5" at 456,212 size 75x75; Picture "Graphic_14"
      HorizontalMovement <- "Machining Center part after maching move"
   Button "Button_5" at 69,129 size 190x62; TextOn 'Main Screen'; TextOff 'Main Screen'
      on Click: ActivateScreen("Main Screen", 0)
   Button "Button_6" at 579,12 size 210x53; TextOn 'Stopped'; TextOff 'Emergency Stop'
      on Release: ResetBit("HMI_AREA_POINTER_Stop PB")
      on Press: SetBit("HMI_AREA_POINTER_Stop PB")
   Button "Button_7" at 514,111 size 192x32; TextOn 'Assembly'; TextOff 'Assembly'
      on Click: ActivateScreen("Assembly", 0)
   Button "Button_8" at 508,159 size 192x32; TextOn 'Pick&Place'; TextOff 'Pick&Place'
      on Click: ActivateScreen("Pick&Place", 0)
   TextField "Text field_2" at 319,311 size 21x32; Text 'Text'
   Circle "Circle_4" at 77,368 size 48x48
      Appearance <- "Bases_raw_conveyor"
   Circle "Circle_8" at 246,368 size 48x48
      Appearance <- "Exit_Conveyor"
   TextField "Text field_1" at 51,318 size 118x32; Text 'Working'
   TextField "Text field_4" at 222,320 size 118x32; Text 'Finished'
   TextField "Text field_5" at 389,317 size 76x32; Text 'Error'
   Circle "Circle_1" at 698,317 size 48x48
      Appearance <- "Lids_center_busy"
   TextField "Text field_6" at 498,322 size 199x32; Text 'Leds Machining'
   TextField "Text field_7" at 498,378 size 202x32; Text 'Base Machining'
   Circle "Circle_2" at 700,372 size 48x48
      Appearance <- "bases_center_busy"
   Button "Button_9" at 235,21 size 279x35; TextOn 'Started'; TextOff 'Machining Center Station'
      on Release: ResetBit("HMI_AREA_POINTER_Start PB")
      on Press: SetBit("HMI_AREA_POINTER_Start PB")

screen "Main Screen" 800x420
   Button "Button_3" at 0,49 size 209x44; TextOn 'Started'; TextOff 'Start Whole System'
      on Release: ResetBit("HMI_AREA_POINTER_Start PB")
      on Press: SetBit("HMI_AREA_POINTER_Start PB")
   Button "Button_7" at 206,5 size 277x35; TextOn 'Started'; TextOff 'Main Screen Production line'
      on Release: ResetBit("HMI_AREA_POINTER_Start PB")
      on Press: SetBit("HMI_AREA_POINTER_Start PB")
   Button "Button_4" at 3,106 size 210x40; TextOn 'Stopped'; TextOff 'Stop Whole System'
      on Release: ResetBit("HMI_AREA_POINTER_Stop PB")
      on Press: SetBit("HMI_AREA_POINTER_Stop PB")
   TextField "Text field_1" at 561,14 size 187x32; Text 'Feeding State'
   TextField "Text field_2" at 487,71 size 263x32; Text 'Machining Lid State'
   TextField "Text field_3" at 483,133 size 286x32; Text 'Machining Base State'
   TextField "Text field_4" at 470,320 size 280x32; Text 'Assembly Green state'
   TextField "Text field_5" at 487,377 size 261x32; Text 'Assembly Blue state'
   TextField "Text field_6" at 444,193 size 314x32; Text 'Green Material Detected'
   TextField "Text field_7" at 461,259 size 295x32; Text 'Blue Material Detected'
   Button "Button_1" at 107,429 size 192x32; TextOn 'Alarm'; TextOff 'Alarm'
      on Click: ActivateScreen("Alarm", 0)
   Button "Button_2" at 0,333 size 192x32; TextOn 'Pick&Place'; TextOff 'Pick&Place'
      on Click: ActivateScreen("Pick&Place", 0)
   Button "Button_5" at 0,381 size 192x32; TextOn 'Sorting'; TextOff 'Sorting'
      on Click: ActivateScreen("Sorting", 0)
   Button "Button_6" at 206,334 size 192x32; TextOn 'Machine Center'; TextOff 'Machine Center'
      on Click: ActivateScreen("Machine Center", 0)
   Button "Button_8" at 206,378 size 192x32; TextOn 'Assembly'; TextOff 'Assembly'
      on Click: ActivateScreen("Assembly", 0)
   TextField "Text field_8" at 138,287 size 136x39; Text 'Screens'
   TextField "Text field_9" at 627,437 size 87x32; Text 'Alarm'
   TextField "Text field_10" at 3,249 size 310x32; Text 'Current Green Products'
   TextField "Text field_11" at 0,207 size 290x32; Text 'Current blue Products'
   IOField "I/O field_1" at 297,206 size 96x32; FormatPattern 99
   IOField "I/O field_2" at 301,250 size 96x32; FormatPattern 99
   IOField "I/O field_3" at 340,80 size 71x29; FormatPattern 99
   TextField "Text field_12" at 279,56 size 233x25; Text 'Required blue Products'
   TextField "Text field_13" at 271,119 size 248x25; Text 'Required Green Products'
   IOField "I/O field_4" at 339,146 size 77x29; FormatPattern 99
   GraphicView "Graphic view_1" at 213,46 size 59x58; Picture "image-removebg-preview"
      Appearance <- "s1"
   GraphicView "Graphic view_2" at 216,104 size 51x52; Picture "off"
   Circle "Circle_7" at 747,370 size 43x43
      Appearance <- "S2(7) Blue Assembler"
   Circle "Circle_6" at 747,316 size 41x41
      Appearance <- "S2(8) Green"
   Circle "Circle_8" at 745,193 size 43x43
      Appearance <- "bases Sorter  Belt"
   Circle "Circle_9" at 745,250 size 43x43
      Appearance <- "LID sorter Belt"
   Circle "Circle_3" at 743,1 size 45x45
      Appearance <- "HMI Entry_conveyor"
   Circle "Circle_4" at 744,61 size 44x44
      Appearance <- "Lids_center_busy"
   Circle "Circle_5" at 745,133 size 43x43
      Appearance <- "bases_center_busy"

screen "Pick&Place" 800x420
   GraphicView "Graphic view_1" at 285,177 size 330x46; Picture "Graphic_7"
   GraphicView "Graphic view_2" at 230,218 size 332x53; Picture "Graphic_7"
   GraphicView "Graphic view_3" at 533,150 size 55x48; Picture "Graphic_9"
      Visibility <- "HMI_Box_Pick_and_place1"
      HorizontalMovement <- "HMI_Box_Pick_and_place1"
   GraphicView "Graphic view_4" at 271,198 size 55x48; Picture "Graphic_9"
      Visibility <- "HMI_Box_Pick_and_place2"
      HorizontalMovement <- "HMI_Box_Pick_and_place2"
   GraphicView "Graphic view_6" at 344,68 size 37x78; Picture "Graphic_10"
      Appearance <- "HMI Grab"
   Button "Button_1" at 135,113 size 99x33; TextOn 'Alarm'; TextOff 'Alarm'
      on Click: ActivateScreen("Alarm", 0)
   Button "Button_2" at 93,164 size 192x32; TextOn 'Sorting'; TextOff 'Sorting'
      on Click: ActivateScreen("Sorting", 0)
   Button "Button_7" at 256,0 size 242x35; TextOn 'Started'; TextOff 'Pick and place Station'
      on Release: ResetBit("HMI_AREA_POINTER_Start PB")
      on Press: SetBit("HMI_AREA_POINTER_Start PB")
   Circle "Circle_2" at 407,309 size 48x48
      Appearance <- "HMI Entry_conveyor"
   TextField "Text field_6" at 120,317 size 240x32; Text 'Feeding 1 Working'
   TextField "Text field_7" at 120,373 size 240x32; Text 'Feeding 2 Working'
   Circle "Circle_3" at 407,365 size 48x48
      Appearance <- "Exit conveyor"
   Button "Button_5" at 75,28 size 169x45; TextOn 'Stopped'; TextOff 'Emergency Stop'
      on Release: ResetBit("HMI_AREA_POINTER_Stop PB")
      on Press: SetBit("HMI_AREA_POINTER_Stop PB")

screen "Sorting" 800x420
   Button "Button_4" at 33,37 size 169x45; TextOn 'Stopped'; TextOff 'Emergency Stop'
      on Release: ResetBit("HMI_AREA_POINTER_Stop PB")
      on Press: SetBit("HMI_AREA_POINTER_Stop PB")
   Button "Button_1" at 281,126 size 99x33; TextOn 'Alarm'; TextOff 'Alarm'
   GraphicView "Graphic view_5" at 350,178 size 330x46; Picture "Graphic_7"
   GraphicView "Graphic view_7" at 572,151 size 55x48; Picture "Graphic_9"
      Visibility <- "HMI_Box_Pick_and_place1"
   GraphicView "Graphic view_8" at 584,58 size 37x78; Picture "Graphic_10"
   GraphicView "Graphic view_9" at 268,220 size 189x85; Picture "Graphic_12"
   GraphicView "Graphic view_10" at 485,227 size 189x85; Picture "Graphic_12"
   Button "Button_2" at 60,227 size 192x32; TextOn 'Pick&Place'; TextOff 'Pick&Place'
      on Click: ActivateScreen("Pick&Place", 0)
   Button "Button_5" at 64,280 size 192x32; TextOn 'Assembly'; TextOff 'Assembly'
      on Click: ActivateScreen("Assembly", 0)
   Button "Button_6" at 65,178 size 192x32; TextOn 'Machine Center'; TextOff 'Machine Center'
      on Click: ActivateScreen("Machine Center", 0)
   Button "Button_7" at 260,18 size 242x35; TextOn 'Started'; TextOff 'Sorting Station'
      on Release: ResetBit("HMI_AREA_POINTER_Start PB")
      on Press: SetBit("HMI_AREA_POINTER_Start PB")
   Button "Button_3" at 62,126 size 192x32; TextOn 'Main Screen'; TextOff 'Main Screen'
      on Click: ActivateScreen("Main Screen", 0)
   Button "Button_8" at 488,316 size 192x32; TextOn 'Assembly'; TextOff 'Blue Part Sorted'
      on Click: ActivateScreen("Assembly", 0)
   Button "Button_9" at 266,315 size 192x32; TextOn 'Assembly'; TextOff 'Green Part Sorted'
      on Click: ActivateScreen("Assembly", 0)
   Circle "Circle_1" at 336,353 size 48x48
      Appearance <- "bases Sorter  Belt"
   Circle "Circle_2" at 566,354 size 48x48
      Appearance <- "LID sorter Belt"
   GraphicView "Graphic view_1" at 390,182 size 55x48; Picture "Graphic_9"
      DiagonalMovement <- "HMI Green part sorted move HMI"
      Visibility <- "HMI_Box_Pick_and_place1"
   GraphicView "Graphic view_2" at 608,194 size 55x48; Picture "Graphic_9"
      DiagonalMovement <- "HMI Blue part sorted move HMI"
      Visibility <- "HMI_Box_Pick_and_place1"
*)